C01742=50.626,-85.269,61.037,-178.4250,1.8965,-10229.3015
C01743=46.265,-88.593,61.359,-179.8629,0.0736,-10232.4256
C01744=41.009,-91.197,61.571,-179.9828,0.0078,-10235.7877
C01745=35.488,-93.484,61.571,-179.9823,0.0066,-10239.2124
C01746=29.931,-95.359,61.359,-179.8510,0.0449,-10242.5741
C01747=24.496,-96.092,61.037,-177.5461,-0.2275,-10245.6986
C01748=19.672,-94.474,60.719,-175.8447,-2.5954,-10248.2376
C01749=16.396,-90.884,60.330,-176.4208,-7.1953,-10249.7735
C01750=15.041,-85.905,59.597,-178.1039,-7.6987,-10250.0688
C01751=13.963,-80.549,58.128,-178.6435,-5.7936,-10250.1656
C01752=12.951,-75.822,56.240,-179.3107,-2.5537,-10250.3070
C01753=11.825,-72.328,54.436,178.2362,4.4065,-10250.7148
C01754=9.959,-70.362,53.146,152.3999,15.9321,-10251.9439
C01755=6.412,-69.984,52.637,141.4077,0.6880,-10254.7651
C01756=3.072,-70.158,52.615,141.0087,-2.3123,-10257.4928
C01757=0.000,-70.224,52.630,140.9842,-0.0003,-10260.0000
C01758=0.000,-70.224,52.630,140.9842,-0.0003,-10260.0000
C01759=-3.071,-70.158,52.615,141.0086,2.3125,-10262.5064
C01760=-6.412,-69.984,52.637,141.4081,-0.6906,-10265.2349
C01761=-9.959,-70.362,53.146,152.3995,-15.9318,-10268.0561
C01762=-11.825,-72.328,54.436,178.2362,-4.4065,-10269.2852
C01763=-12.951,-75.822,56.240,-179.3107,2.5537,-10269.6930
C01764=-13.963,-80.549,58.128,-178.6435,5.7936,-10269.8344
C01765=-15.041,-85.905,59.597,-178.1039,7.6987,-10269.9312
C01766=-16.396,-90.884,60.330,-176.4208,7.1953,-10270.2265
C01767=-19.672,-94.474,60.719,-175.8447,2.5954,-10271.7624
C01768=-24.496,-96.092,61.037,-177.5461,0.2275,-10274.3014
C01769=-29.931,-95.359,61.359,-179.8510,-0.0449,-10277.4259
C01770=-35.488,-93.484,61.571,-179.9823,-0.0066,-10280.7876
C01771=-41.009,-91.197,61.571,-179.9828,-0.0078,-10284.2123
C01772=-46.265,-88.593,61.359,-179.8629,-0.0736,-10287.5744
C01773=-50.626,-85.269,61.037,-178.4250,-1.8965,-10290.6985
C01774=-52.893,-80.714,60.719,-178.8932,-4.7688,-10293.2374
C01775=-52.671,-75.858,60.330,177.4212,-7.6040,-10294.7737
C01776=-50.109,-71.379,59.597,175.8716,-6.7862,-10295.0694
C01777=-47.084,-66.830,58.128,176.8518,-5.0569,-10295.1660
C01778=-44.457,-62.772,56.240,178.6807,-2.2931,-10295.3073
C01779=-42.782,-59.505,54.436,-178.1262,4.3612,-10295.7148
C01780=-42.712,-56.796,53.146,170.4736,29.7489,-10296.9441
C01781=-44.952,-54.020,52.637,150.9334,29.8046,-10299.7651
C01782=-47.437,-51.781,52.615,148.9950,28.5406,-10302.4931
C01783=-49.656,-49.656,52.630,150.1903,29.8094,-10305.0000
C01784=-51.781,-47.437,52.615,151.4594,31.0052,-10307.5069
C01785=-54.020,-44.952,52.637,150.1944,29.0648,-10310.2349
C01786=-56.796,-42.711,53.146,150.2510,9.5269,-10313.0566
C01787=-59.505,-42.782,54.436,175.6388,-1.8738,-10314.2852
C01788=-62.772,-44.457,56.240,-177.7069,1.3193,-10314.6927
C01789=-66.830,-47.084,58.128,-174.9431,3.1482,-10314.8340
C01790=-71.379,-50.109,59.597,-173.2138,4.1284,-10314.9306
C01791=-75.858,-52.671,60.330,-172.3960,2.5788,-10315.2263
C01792=-80.714,-52.893,60.719,-175.2312,-1.1068,-10316.7626
C01793=-85.269,-50.626,61.037,-178.1035,-1.5750,-10319.3015
C01794=-88.593,-46.265,61.359,-179.9264,-0.1371,-10322.4256
C01795=-91.197,-41.009,61.571,-179.9922,-0.0172,-10325.7877
C01796=-93.484,-35.488,61.571,-179.9934,-0.0177,-10329.2124
C01797=-95.359,-29.931,61.359,-179.9551,-0.1490,-10332.5741
C01798=-96.092,-24.496,61.037,179.7725,-2.4539,-10335.6986
C01799=-94.474,-19.672,60.719,177.4046,-4.1553,-10338.2376
C01800=-90.884,-16.396,60.330,172.8047,-3.5792,-10339.7735
C01801=-85.905,-15.041,59.597,172.3013,-1.8961,-10340.0688
C01802=-80.549,-13.963,58.128,174.2064,-1.3565,-10340.1656
C01803=-75.822,-12.951,56.240,177.4463,-0.6893,-10340.3070
C01804=-72.328,-11.825,54.436,-175.5935,1.7638,-10340.7148
C01805=-70.362,-9.959,53.146,-164.0679,27.6001,-10341.9439
C01806=-69.984,-6.412,52.637,-179.3120,38.5923,-10344.7651
C01807=-70.158,-3.072,52.615,177.6877,38.9913,-10347.4928
C01808=-70.224,0.000,52.630,179.9997,39.0158,-10350.0000
C01809=-70.158,3.071,52.615,-177.6875,38.9914,-10352.5064
C01810=-69.984,6.412,52.637,179.3094,38.5919,-10355.2349
C01811=-70.362,9.959,53.146,164.0682,27.6005,-10358.0561
C01812=-72.328,11.825,54.436,175.5935,1.7638,-10359.2852
C01813=-75.822,12.951,56.240,-177.4463,-0.6893,-10359.6930
C01814=-80.549,13.963,58.128,-174.2064,-1.3565,-10359.8344
C01815=-85.905,15.041,59.597,-172.3013,-1.8961,-10359.9312
C01816=-90.884,16.396,60.330,-172.8047,-3.5792,-10360.2265
C01817=-94.474,19.672,60.719,-177.4046,-4.1553,-10361.7624
C01818=-96.092,24.496,61.037,-179.7725,-2.4539,-10364.3014
C01819=-95.359,29.931,61.359,179.9551,-0.1490,-10367.4259
C01820=-93.484,35.488,61.571,179.9934,-0.0177,-10370.7876
C01821=-91.197,41.009,61.571,179.9922,-0.0172,-10374.2123
C01822=-88.593,46.265,61.359,179.9264,-0.1371,-10377.5744
C01823=-85.269,50.626,61.037,178.1035,-1.5750,-10380.6985
C01824=-80.714,52.893,60.719,175.2312,-1.1068,-10383.2374
C01825=-75.858,52.671,60.330,172.3960,2.5788,-10384.7737
C01826=-71.379,50.109,59.597,173.2138,4.1284,-10385.0694
C01827=-66.830,47.084,58.128,174.9431,3.1482,-10385.1660
C01828=-62.772,44.457,56.240,177.7069,1.3193,-10385.3073
C01829=-59.505,42.782,54.436,-175.6388,-1.8738,-10385.7148
C01830=-56.796,42.712,53.146,-150.2511,9.5264,-10386.9441
C01831=-54.020,44.952,52.637,-150.1954,29.0666,-10389.7651
C01832=-51.781,47.437,52.615,-151.4594,31.0050,-10392.4931
C01833=-49.656,49.656,52.630,-150.1906,29.8097,-10395.0000
C01834=-47.437,51.781,52.615,-148.9948,28.5406,-10397.5069
C01835=-44.952,54.020,52.637,-150.9352,29.8056,-10400.2349
C01836=-42.711,56.796,53.146,-170.4731,29.7490,-10403.0566
C01837=-42.782,59.505,54.436,178.1262,4.3612,-10404.2852
C01838=-44.457,62.772,56.240,-178.6807,-2.2931,-10404.6927
C01839=-47.084,66.830,58.128,-176.8518,-5.0569,-10404.8340
C01840=-50.109,71.379,59.597,-175.8716,-6.7862,-10404.9306
C01841=-52.671,75.858,60.330,-177.4212,-7.6040,-10405.2263
C01842=-52.893,80.714,60.719,178.8932,-4.7688,-10406.7626
C01843=-50.626,85.269,61.037,178.4250,-1.8965,-10409.3015
C01844=-46.265,88.593,61.359,179.8629,-0.0736,-10412.4256
C01845=-41.009,91.197,61.571,179.9828,-0.0078,-10415.7877
C01846=-35.488,93.484,61.571,179.9823,-0.0066,-10419.2124
C01847=-29.931,95.359,61.359,179.8510,-0.0449,-10422.5741
C01848=-24.496,96.092,61.037,177.5461,0.2275,-10425.6986
C01849=-19.672,94.474,60.719,175.8447,2.5954,-10428.2376
C01850=-16.396,90.884,60.330,176.4208,7.1953,-10429.7735
C01851=-15.041,85.905,59.597,178.1039,7.6987,-10430.0688
C01852=-13.963,80.549,58.128,178.6435,5.7936,-10430.1656
C01853=-12.951,75.822,56.240,179.3107,2.5537,-10430.3070
C01854=-11.825,72.328,54.436,-178.2362,-4.4065,-10430.7148
C01855=-9.959,70.362,53.146,-152.3995,-15.9318,-10431.9439
C01856=-6.412,69.984,52.637,-141.4081,-0.6906,-10434.7651
C01857=-3.071,70.158,52.615,-141.0086,2.3125,-10437.4936
C01858=0.000,70.224,52.630,-140.9842,-0.0003,-10440.0000
C01859=0.000,68.843,54.342,-141.2235,-0.0004,-10440.0000
C01860=2.945,68.781,54.326,-141.2470,-2.2595,-10442.4517
C01861=6.200,68.619,54.350,-141.6907,1.0492,-10445.1629
C01862=9.699,69.044,54.888,-153.6475,16.2162,-10447.9963
C01863=11.507,71.127,56.252,-178.7377,3.4210,-10449.1897
C01864=12.586,74.809,58.158,179.2393,-3.0039,-10449.5501
C01865=13.569,79.780,60.151,178.6797,-5.9734,-10449.6525
C01866=14.621,85.405,61.698,178.2099,-7.7575,-10449.7146
C01867=15.942,90.636,62.469,176.5679,-7.2955,-10449.9757
C01868=19.246,94.423,62.877,175.8470,-2.7058,-10451.5206
C01869=24.159,96.154,63.210,177.5359,-0.2528,-10454.1038
C01870=29.718,95.429,63.547,179.8486,0.0454,-10457.2974
C01871=35.416,93.512,63.770,179.9821,0.0067,-10460.7433
C01872=41.080,91.166,63.770,179.9826,0.0079,-10464.2566
C01873=46.465,88.493,63.547,179.8609,0.0749,-10467.7026
C01874=50.908,85.074,63.210,178.4357,1.9214,-10470.8962
C01875=53.158,80.376,62.877,178.9730,4.8449,-10473.4793
C01876=52.817,75.362,62.469,-177.2451,7.5721,-10475.0245
C01877=50.052,70.729,61.698,-175.7549,6.7538,-10475.2855
C01878=46.818,66.007,60.151,-176.6982,5.1590,-10475.3476
C01879=43.998,61.798,58.158,-178.4123,2.6620,-10475.4495
C01880=42.158,58.431,56.252,178.4711,-3.3109,-10475.8105
C01881=41.963,55.679,54.888,-171.7704,-29.0710,-10477.0038
C01882=44.137,52.905,54.350,-151.3798,-29.7512,-10479.8372
C01883=46.553,50.718,54.326,-149.2273,-28.3546,-10482.5482
C01884=48.679,48.679,54.342,-150.4011,-29.5986,-10485.0000
C01885=50.718,46.553,54.326,-151.6456,-30.7729,-10487.4518
C01886=52.905,44.137,54.350,-150.2477,-28.6184,-10490.1628
C01887=55.680,41.963,54.888,-150.9289,-8.2300,-10492.9966
C01888=58.431,42.158,56.252,-176.6891,1.5289,-10494.1895
C01889=61.798,43.998,58.158,177.3380,-1.5877,-10494.5505
C01890=66.007,46.818,60.151,174.8410,-3.3018,-10494.6524
C01891=70.729,50.052,61.698,173.2462,-4.2451,-10494.7145
C01892=75.362,52.817,62.469,172.4279,-2.7549,-10494.9755
C01893=80.376,53.158,62.877,175.1551,1.0270,-10496.5207
C01894=85.074,50.908,63.210,178.0786,1.5643,-10499.1038
C01895=88.493,46.465,63.547,179.9251,0.1391,-10502.2974
C01896=91.166,41.080,63.770,179.9921,0.0174,-10505.7434
C01897=93.512,35.416,63.770,179.9933,0.0179,-10509.2567
C01898=95.429,29.718,63.547,179.9546,0.1514,-10512.7026
C01899=96.154,24.159,63.210,-179.7472,2.4641,-10515.8962
C01900=94.423,19.246,62.877,-177.2942,4.1530,-10518.4794
C01901=90.636,15.942,62.469,-172.7045,3.4321,-10520.0243
C01902=85.405,14.621,61.698,-172.2425,1.7901,-10520.2854
C01903=79.780,13.569,60.151,-174.0266,1.3203,-10520.3475
C01904=74.809,12.586,58.158,-176.9961,0.7607,-10520.4499
C01905=71.127,11.507,56.252,176.5790,-1.2623,-10520.8103
C01906=69.044,9.699,54.888,163.7838,-26.3525,-10522.0037
C01907=68.619,6.200,54.350,178.9508,-38.3093,-10524.8371
C01908=68.781,2.945,54.326,-177.7405,-38.7530,-10527.5483
C01909=68.843,0.000,54.342,-179.9996,-38.7765,-10530.0000
C01910=68.781,-2.945,54.326,177.7401,-38.7530,-10532.4517
C01911=68.619,-6.200,54.350,-178.9482,-38.3089,-10535.1629
C01912=69.044,-9.699,54.888,-163.7840,-26.3528,-10537.9963
C01913=71.127,-11.507,56.252,-176.5790,-1.2623,-10539.1897
C01914=74.809,-12.586,58.158,176.9961,0.7607,-10539.5501
C01915=79.780,-13.569,60.151,174.0266,1.3203,-10539.6525
C01916=85.405,-14.621,61.698,172.2425,1.7901,-10539.7146
C01917=90.636,-15.942,62.469,172.7045,3.4321,-10539.9757
C01918=94.423,-19.246,62.877,177.2942,4.1530,-10541.5206
C01919=96.154,-24.159,63.210,179.7472,2.4641,-10544.1038
C01920=95.429,-29.718,63.547,-179.9546,0.1514,-10547.2974
C01921=93.512,-35.416,63.770,-179.9933,0.0179,-10550.7433
C01922=91.166,-41.080,63.770,-179.9921,0.0174,-10554.2566
C01923=88.493,-46.465,63.547,-179.9251,0.1391,-10557.7026
C01924=85.074,-50.908,63.210,-178.0786,1.5643,-10560.8962
C01925=80.376,-53.158,62.877,-175.1551,1.0270,-10563.4793
C01926=75.362,-52.817,62.469,-172.4279,-2.7549,-10565.0245
C01927=70.729,-50.052,61.698,-173.2462,-4.2451,-10565.2855
C01928=66.007,-46.818,60.151,-174.8410,-3.3018,-10565.3476
C01929=61.798,-43.998,58.158,-177.3380,-1.5877,-10565.4495
C01930=58.431,-42.158,56.252,176.6891,1.5289,-10565.8105
C01931=55.679,-41.963,54.888,150.9290,-8.2296,-10567.0038
C01932=52.905,-44.137,54.350,150.2488,-28.6202,-10569.8372
C01933=50.718,-46.553,54.326,151.6454,-30.7727,-10572.5482
C01934=48.679,-48.679,54.342,150.4014,-29.5989,-10575.0000
C01935=46.553,-50.718,54.326,149.2271,-28.3544,-10577.4518
C01936=44.137,-52.905,54.350,151.3816,-29.7523,-10580.1628
C01937=41.963,-55.680,54.888,171.7700,-29.0711,-10582.9966
C01938=42.158,-58.431,56.252,-178.4711,-3.3109,-10584.1895
C01939=43.998,-61.798,58.158,178.4123,2.6620,-10584.5505
C01940=46.818,-66.007,60.151,176.6982,5.1590,-10584.6524
C01941=50.052,-70.729,61.698,175.7549,6.7538,-10584.7145
C01942=52.817,-75.362,62.469,177.2451,7.5721,-10584.9755
C01943=53.158,-80.376,62.877,-178.9730,4.8449,-10586.5207
C01944=50.908,-85.074,63.210,-178.4357,1.9214,-10589.1038
C01945=46.465,-88.493,63.547,-179.8609,0.0749,-10592.2974
C01946=41.080,-91.166,63.770,-179.9826,0.0079,-10595.7434
C01947=35.416,-93.512,63.770,-179.9821,0.0067,-10599.2567
C01948=29.718,-95.429,63.547,-179.8486,0.0454,-10602.7026
C01949=24.159,-96.154,63.210,-177.5359,-0.2528,-10605.8962
C01950=19.246,-94.423,62.877,-175.8470,-2.7058,-10608.4794
C01951=15.942,-90.636,62.469,-176.5679,-7.2955,-10610.0243
C01952=14.621,-85.405,61.698,-178.2099,-7.7575,-10610.2854
C01953=13.569,-79.780,60.151,-178.6797,-5.9734,-10610.3475
C01954=12.586,-74.809,58.158,-179.2393,-3.0039,-10610.4499
C01955=11.507,-71.127,56.252,178.7377,3.4210,-10610.8103
C01956=9.699,-69.044,54.888,153.6475,16.2162,-10612.0037
C01957=6.200,-68.619,54.350,141.6907,1.0492,-10614.8371
C01958=2.945,-68.781,54.326,141.2470,-2.2595,-10617.5483
C01959=0.000,-68.843,54.342,141.2235,-0.0004,-10620.0000
C01960=0.000,-68.843,54.342,141.2235,-0.0004,-10620.0000
C01961=-2.945,-68.781,54.326,141.2470,2.2599,-10622.4517
C01962=-6.200,-68.619,54.350,141.6911,-1.0518,-10625.1629
C01963=-9.699,-69.044,54.888,153.6472,-16.2160,-10627.9963
C01964=-11.507,-71.127,56.252,178.7377,-3.4210,-10629.1897
C01965=-12.586,-74.809,58.158,-179.2393,3.0039,-10629.5501
C01966=-13.569,-79.780,60.151,-178.6797,5.9734,-10629.6525
C01967=-14.621,-85.405,61.698,-178.2099,7.7575,-10629.7146
C01968=-15.942,-90.636,62.469,-176.5679,7.2955,-10629.9757
C01969=-19.246,-94.423,62.877,-175.8470,2.7058,-10631.5206
C01970=-24.159,-96.154,63.210,-177.5359,0.2528,-10634.1038
C01971=-29.718,-95.429,63.547,-179.8486,-0.0454,-10637.2974
C01972=-35.416,-93.512,63.770,-179.9821,-0.0067,-10640.7433
C01973=-41.080,-91.166,63.770,-179.9826,-0.0079,-10644.2566
C01974=-46.465,-88.493,63.547,-179.8609,-0.0749,-10647.7026
C01975=-50.908,-85.074,63.210,-178.4357,-1.9214,-10650.8962
C01976=-53.158,-80.376,62.877,-178.9730,-4.8449,-10653.4793
C01977=-52.817,-75.362,62.469,177.2451,-7.5721,-10655.0245
C01978=-50.052,-70.729,61.698,175.7549,-6.7538,-10655.2855
C01979=-46.818,-66.007,60.151,176.6982,-5.1590,-10655.3476
C01980=-43.998,-61.798,58.158,178.4123,-2.6620,-10655.4495
C01981=-42.158,-58.431,56.252,-178.4711,3.3109,-10655.8105
C01982=-41.963,-55.679,54.888,171.7704,29.0710,-10657.0038
C01983=-44.137,-52.905,54.350,151.3798,29.7512,-10659.8372
C01984=-46.553,-50.718,54.326,149.2273,28.3546,-10662.5482
C01985=-48.679,-48.679,54.342,150.4011,29.5986,-10665.0000
C01986=-50.718,-46.553,54.326,151.6456,30.7729,-10667.4518
C01987=-52.905,-44.137,54.350,150.2477,28.6184,-10670.1628
C01988=-55.680,-41.963,54.888,150.9289,8.2300,-10672.9966
C01989=-58.431,-42.158,56.252,176.6891,-1.5289,-10674.1895
C01990=-61.798,-43.998,58.158,-177.3380,1.5877,-10674.5505
C01991=-66.007,-46.818,60.151,-174.8410,3.3018,-10674.6524
C01992=-70.729,-50.052,61.698,-173.2462,4.2451,-10674.7145
C01993=-75.362,-52.817,62.469,-172.4279,2.7549,-10674.9755
C01994=-80.376,-53.158,62.877,-175.1551,-1.0270,-10676.5207
C01995=-85.074,-50.908,63.210,-178.0786,-1.5643,-10679.1038
C01996=-88.493,-46.465,63.547,-179.9251,-0.1391,-10682.2974
C01997=-91.166,-41.080,63.770,-179.9921,-0.0174,-10685.7434
C01998=-93.512,-35.416,63.770,-179.9933,-0.0179,-10689.2567
C01999=-95.429,-29.718,63.547,-179.9546,-0.1514,-10692.7026
///TOOL 0
///POSTYPE ANGLE
///ANGLE
EC00000=0.0000,7126.2037
EC00001=0.0000,7128.6701
EC00002=0.0000,7131.2180
EC00003=0.0000,7133.7821
EC00004=0.0000,7136.3297
EC00005=0.0000,7138.7961
EC00006=0.0000,7140.9450
EC00007=0.0000,7142.4587
EC00008=0.0000,7143.1487
EC00009=0.0000,7143.6320
EC00010=0.0000,7144.1614
EC00011=0.0000,7144.9722
EC00012=0.0000,7146.4919
EC00013=0.0000,7149.2230
EC00014=0.0000,7152.0820
EC00015=0.0000,7155.0000
EC00016=0.0000,7157.9180
EC00017=0.0000,7160.7770
EC00018=0.0000,7163.5081
EC00019=0.0000,7165.0278
EC00020=0.0000,7165.8386
EC00021=0.0000,7166.3680
EC00022=0.0000,7166.8513
EC00023=0.0000,7167.5413
EC00024=0.0000,7169.0550
EC00025=0.0000,7171.2039
EC00026=0.0000,7173.6703
EC00027=0.0000,7176.2179
EC00028=0.0000,7178.7820
EC00029=0.0000,7181.3299
EC00030=0.0000,7183.7963
EC00031=0.0000,7185.9450
EC00032=0.0000,7187.4590
EC00033=0.0000,7188.1488
EC00034=0.0000,7188.6317
EC00035=0.0000,7189.1618
EC00036=0.0000,7189.9720
EC00037=0.0000,7191.4924
EC00038=0.0000,7194.2225
EC00039=0.0000,7197.0820
EC00040=0.0000,7200.0000
EC00041=0.0000,7200.0000
EC00042=0.0000,7202.8792
EC00043=0.0000,7205.7259
EC00044=0.0000,7208.4654
EC00045=0.0000,7209.9566
EC00046=0.0000,7210.7254
EC00047=0.0000,7211.2119
EC00048=0.0000,7211.6495
EC00049=0.0000,7212.2909
EC00050=0.0000,7213.8024
EC00051=0.0000,7215.9922
EC00052=0.0000,7218.5312
EC00053=0.0000,7221.1696
EC00054=0.0000,7223.8303
EC00055=0.0000,7226.4689
EC00056=0.0000,7229.0082
EC00057=0.0000,7231.1977
EC00058=0.0000,7232.7089
EC00059=0.0000,7233.3509
EC00060=0.0000,7233.7878
EC00061=0.0000,7234.2746
EC00062=0.0000,7235.0436
EC00063=0.0000,7236.5348
EC00064=0.0000,7239.2737
EC00065=0.0000,7242.1206
EC00066=0.0000,7245.0000
EC00067=0.0000,7247.8789
EC00068=0.0000,7250.7263
EC00069=0.0000,7253.4652
EC00070=0.0000,7254.9564
EC00071=0.0000,7255.7254
EC00072=0.0000,7256.2122
EC00073=0.0000,7256.6491
EC00074=0.0000,7257.2911
EC00075=0.0000,7258.8023
EC00076=0.0000,7260.9918
EC00077=0.0000,7263.5311
EC00078=0.0000,7266.1697
EC00079=0.0000,7268.8304
EC00080=0.0000,7271.4688
EC00081=0.0000,7274.0078
EC00082=0.0000,7276.1976
EC00083=0.0000,7277.7091
EC00084=0.0000,7278.3505
EC00085=0.0000,7278.7881
EC00086=0.0000,7279.2746
EC00087=0.0000,7280.0434
EC00088=0.0000,7281.5346
EC00089=0.0000,7284.2741
EC00090=0.0000,7287.1208
EC00091=0.0000,7290.0000
EC00092=0.0000,7292.8792
EC00093=0.0000,7295.7266
EC00094=0.0000,7298.4654
EC00095=0.0000,7299.9566
EC00096=0.0000,7300.7254
EC00097=0.0000,7301.2119
EC00098=0.0000,7301.6495
EC00099=0.0000,7302.2909
EC00100=0.0000,7303.8024
EC00101=0.0000,7305.9922
EC00102=0.0000,7308.5312
EC00103=0.0000,7311.1696
EC00104=0.0000,7313.8303
EC00105=0.0000,7316.4689
EC00106=0.0000,7319.0082
EC00107=0.0000,7321.1977
EC00108=0.0000,7322.7089
EC00109=0.0000,7323.3509
EC00110=0.0000,7323.7878
EC00111=0.0000,7324.2746
EC00112=0.0000,7325.0436
EC00113=0.0000,7326.5348
EC00114=0.0000,7329.2737
EC00115=0.0000,7332.1206
EC00116=0.0000,7335.0000
EC00117=0.0000,7337.8789
EC00118=0.0000,7340.7263
EC00119=0.0000,7343.4652
EC00120=0.0000,7344.9564
EC00121=0.0000,7345.7254
EC00122=0.0000,7346.2122
EC00123=0.0000,7346.6491
EC00124=0.0000,7347.2911
EC00125=0.0000,7348.8023
EC00126=0.0000,7350.9918
EC00127=0.0000,7353.5311
EC00128=0.0000,7356.1697
EC00129=0.0000,7358.8304
EC00130=0.0000,7361.4688
EC00131=0.0000,7364.0078
EC00132=0.0000,7366.1976
EC00133=0.0000,7367.7091
EC00134=0.0000,7368.3505
EC00135=0.0000,7368.7881
EC00136=0.0000,7369.2746
EC00137=0.0000,7370.0434
EC00138=0.0000,7371.5346
EC00139=0.0000,7374.2741
EC00140=0.0000,7377.1208
EC00141=0.0000,7380.0000
EC00142=0.0000,7380.0000
EC00143=0.0000,7382.8792
EC00144=0.0000,7385.7266
EC00145=0.0000,7388.4654
EC00146=0.0000,7389.9566
EC00147=0.0000,7390.7254
EC00148=0.0000,7391.2119
EC00149=0.0000,7391.6495
EC00150=0.0000,7392.2909
EC00151=0.0000,7393.8024
EC00152=0.0000,7395.9922
EC00153=0.0000,7398.5312
EC00154=0.0000,7401.1696
EC00155=0.0000,7403.8303
EC00156=0.0000,7406.4689
EC00157=0.0000,7409.0082
EC00158=0.0000,7411.1977
EC00159=0.0000,7412.7089
EC00160=0.0000,7413.3509
EC00161=0.0000,7413.7878
EC00162=0.0000,7414.2746
EC00163=0.0000,7415.0436
EC00164=0.0000,7416.5348
EC00165=0.0000,7419.2737
EC00166=0.0000,7422.1206
EC00167=0.0000,7425.0000
EC00168=0.0000,7427.8789
EC00169=0.0000,7430.7263
EC00170=0.0000,7433.4652
EC00171=0.0000,7434.9564
EC00172=0.0000,7435.7254
EC00173=0.0000,7436.2122
EC00174=0.0000,7436.6491
EC00175=0.0000,7437.2911
EC00176=0.0000,7438.8023
EC00177=0.0000,7440.9918
EC00178=0.0000,7443.5311
EC00179=0.0000,7446.1697
EC00180=0.0000,7448.8304
EC00181=0.0000,7451.4688
EC00182=0.0000,7454.0078
EC00183=0.0000,7456.1976
EC00184=0.0000,7457.7091
EC00185=0.0000,7458.3505
EC00186=0.0000,7458.7881
EC00187=0.0000,7459.2746
EC00188=0.0000,7460.0434
EC00189=0.0000,7461.5346
EC00190=0.0000,7464.2741
EC00191=0.0000,7467.1208
EC00192=0.0000,7470.0000
EC00193=0.0000,7472.8792
EC00194=0.0000,7475.7266
EC00195=0.0000,7478.4654
EC00196=0.0000,7479.9566
EC00197=0.0000,7480.7254
EC00198=0.0000,7481.2119
EC00199=0.0000,7481.6495
EC00200=0.0000,7482.2909
EC00201=0.0000,7483.8024
EC00202=0.0000,7485.9922
EC00203=0.0000,7488.5312
EC00204=0.0000,7491.1696
EC00205=0.0000,7493.8303
EC00206=0.0000,7496.4689
EC00207=0.0000,7499.0082
EC00208=0.0000,7501.1977
EC00209=0.0000,7502.7089
EC00210=0.0000,7503.3509
EC00211=0.0000,7503.7878
EC00212=0.0000,7504.2746
EC00213=0.0000,7505.0436
EC00214=0.0000,7506.5348
EC00215=0.0000,7509.2737
EC00216=0.0000,7512.1206
EC00217=0.0000,7515.0000
EC00218=0.0000,7517.8789
EC00219=0.0000,7520.7263
EC00220=0.0000,7523.4652
EC00221=0.0000,7524.9564
EC00222=0.0000,7525.7254
EC00223=0.0000,7526.2122
EC00224=0.0000,7526.6491
EC00225=0.0000,7527.2911
EC00226=0.0000,7528.8023
EC00227=0.0000,7530.9918
EC00228=0.0000,7533.5311
EC00229=0.0000,7536.1697
EC00230=0.0000,7538.8304
EC00231=0.0000,7541.4688
EC00232=0.0000,7544.0078
EC00233=0.0000,7546.1976
EC00234=0.0000,7547.7091
EC00235=0.0000,7548.3505
EC00236=0.0000,7548.7881
EC00237=0.0000,7549.2746
EC00238=0.0000,7550.0434
EC00239=0.0000,7551.5346
EC00240=0.0000,7554.2734
EC00241=0.0000,7557.1208
EC00242=0.0000,7560.0000
EC00243=0.0000,7560.0000
EC00244=0.0000,7562.8388
EC00245=0.0000,7565.6728
EC00246=0.0000,7568.4202
EC00247=0.0000,7569.8823
EC00248=0.0000,7570.6084
EC00249=0.0000,7571.0516
EC00250=0.0000,7571.4429
EC00251=0.0000,7572.0370
EC00252=0.0000,7573.5473
EC00253=0.0000,7575.7781
EC00254=0.0000,7578.3907
EC00255=0.0000,7581.1209
EC00256=0.0000,7583.8793
EC00257=0.0000,7586.6097
EC00258=0.0000,7589.2218
EC00259=0.0000,7591.4529
EC00260=0.0000,7592.9628
EC00261=0.0000,7593.5569
EC00262=0.0000,7593.9481
EC00263=0.0000,7594.3909
EC00264=0.0000,7595.1173
EC00265=0.0000,7596.5793
EC00266=0.0000,7599.3269
EC00267=0.0000,7602.1606
EC00268=0.0000,7605.0000
EC00269=0.0000,7607.8388
EC00270=0.0000,7610.6731
EC00271=0.0000,7613.4207
EC00272=0.0000,7614.8827
EC00273=0.0000,7615.6091
EC00274=0.0000,7616.0519
EC00275=0.0000,7616.4431
EC00276=0.0000,7617.0372
EC00277=0.0000,7618.5471
EC00278=0.0000,7620.7782
EC00279=0.0000,7623.3903
EC00280=0.0000,7626.1207
EC00281=0.0000,7628.8791
EC00282=0.0000,7631.6093
EC00283=0.0000,7634.2219
EC00284=0.0000,7636.4527
EC00285=0.0000,7637.9630
EC00286=0.0000,7638.5571
EC00287=0.0000,7638.9484
EC00288=0.0000,7639.3916
EC00289=0.0000,7640.1177
EC00290=0.0000,7641.5798
EC00291=0.0000,7644.3272
EC00292=0.0000,7647.1612
EC00293=0.0000,7650.0000
EC00294=0.0000,7652.8388
EC00295=0.0000,7655.6728
EC00296=0.0000,7658.4209
EC00297=0.0000,7659.8823
EC00298=0.0000,7660.6084
EC00299=0.0000,7661.0516
EC00300=0.0000,7661.4429
EC00301=0.0000,7662.0370
EC00302=0.0000,7663.5473
EC00303=0.0000,7665.7781
EC00304=0.0000,7668.3907
EC00305=0.0000,7671.1209
EC00306=0.0000,7673.8793
EC00307=0.0000,7676.6097
EC00308=0.0000,7679.2218
EC00309=0.0000,7681.4529
EC00310=0.0000,7682.9628
EC00311=0.0000,7683.5569
EC00312=0.0000,7683.9481
EC00313=0.0000,7684.3909
EC00314=0.0000,7685.1173
EC00315=0.0000,7686.5793
EC00316=0.0000,7689.3269
EC00317=0.0000,7692.1606
EC00318=0.0000,7695.0000
EC00319=0.0000,7697.8388
EC00320=0.0000,7700.6731
EC00321=0.0000,7703.4207
EC00322=0.0000,7704.8827
EC00323=0.0000,7705.6091
EC00324=0.0000,7706.0519
EC00325=0.0000,7706.4431
EC00326=0.0000,7707.0372
EC00327=0.0000,7708.5471
EC00328=0.0000,7710.7782
EC00329=0.0000,7713.3903
EC00330=0.0000,7716.1207
EC00331=0.0000,7718.8791
EC00332=0.0000,7721.6093
EC00333=0.0000,7724.2219
EC00334=0.0000,7726.4527
EC00335=0.0000,7727.9630
EC00336=0.0000,7728.5571
EC00337=0.0000,7728.9484
EC00338=0.0000,7729.3916
EC00339=0.0000,7730.1177
EC00340=0.0000,7731.5798
EC00341=0.0000,7734.3272
EC00342=0.0000,7737.1612
EC00343=0.0000,7740.0000
EC00344=0.0000,7740.0000
EC00345=0.0000,7742.8388
EC00346=0.0000,7745.6728
EC00347=0.0000,7748.4209
EC00348=0.0000,7749.8823
EC00349=0.0000,7750.6084
EC00350=0.0000,7751.0516
EC00351=0.0000,7751.4429
EC00352=0.0000,7752.0370
EC00353=0.0000,7753.5473
EC00354=0.0000,7755.7781
EC00355=0.0000,7758.3907
EC00356=0.0000,7761.1209
EC00357=0.0000,7763.8793
EC00358=0.0000,7766.6097
EC00359=0.0000,7769.2218
EC00360=0.0000,7771.4529
EC00361=0.0000,7772.9628
EC00362=0.0000,7773.5569
EC00363=0.0000,7773.9481
EC00364=0.0000,7774.3909
EC00365=0.0000,7775.1173
EC00366=0.0000,7776.5793
EC00367=0.0000,7779.3269
EC00368=0.0000,7782.1606
EC00369=0.0000,7785.0000
EC00370=0.0000,7787.8388
EC00371=0.0000,7790.6731
EC00372=0.0000,7793.4207
EC00373=0.0000,7794.8827
EC00374=0.0000,7795.6091
EC00375=0.0000,7796.0519
EC00376=0.0000,7796.4431
EC00377=0.0000,7797.0372
EC00378=0.0000,7798.5471
EC00379=0.0000,7800.7782
EC00380=0.0000,7803.3903
EC00381=0.0000,7806.1207
EC00382=0.0000,7808.8791
EC00383=0.0000,7811.6093
EC00384=0.0000,7814.2219
EC00385=0.0000,7816.4527
EC00386=0.0000,7817.9630
EC00387=0.0000,7818.5571
EC00388=0.0000,7818.9484
EC00389=0.0000,7819.3916
EC00390=0.0000,7820.1177
EC00391=0.0000,7821.5798
EC00392=0.0000,7824.3272
EC00393=0.0000,7827.1612
EC00394=0.0000,7830.0000
EC00395=0.0000,7832.8388
EC00396=0.0000,7835.6728
EC00397=0.0000,7838.4209
EC00398=0.0000,7839.8823
EC00399=0.0000,7840.6084
EC00400=0.0000,7841.0516
EC00401=0.0000,7841.4429
EC00402=0.0000,7842.0370
EC00403=0.0000,7843.5473
EC00404=0.0000,7845.7781
EC00405=0.0000,7848.3907
EC00406=0.0000,7851.1209
EC00407=0.0000,7853.8793
EC00408=0.0000,7856.6097
EC00409=0.0000,7859.2218
EC00410=0.0000,7861.4529
EC00411=0.0000,7862.9628
EC00412=0.0000,7863.5569
EC00413=0.0000,7863.9481
EC00414=0.0000,7864.3909
EC00415=0.0000,7865.1173
EC00416=0.0000,7866.5793
EC00417=0.0000,7869.3269
EC00418=0.0000,7872.1606
EC00419=0.0000,7875.0000
EC00420=0.0000,7877.8388
EC00421=0.0000,7880.6731
EC00422=0.0000,7883.4207
EC00423=0.0000,7884.8827
EC00424=0.0000,7885.6091
EC00425=0.0000,7886.0519
EC00426=0.0000,7886.4431
EC00427=0.0000,7887.0372
EC00428=0.0000,7888.5471
EC00429=0.0000,7890.7782
EC00430=0.0000,7893.3903
EC00431=0.0000,7896.1207
EC00432=0.0000,7898.8791
EC00433=0.0000,7901.6093
EC00434=0.0000,7904.2219
EC00435=0.0000,7906.4527
EC00436=0.0000,7907.9630
EC00437=0.0000,7908.5571
EC00438=0.0000,7908.9484
EC00439=0.0000,7909.3916
EC00440=0.0000,7910.1177
EC00441=0.0000,7911.5791
EC00442=0.0000,7914.3272
EC00443=0.0000,7917.1612
EC00444=0.0000,7920.0000
EC00445=0.0000,7920.0000
EC00446=0.0000,7922.7966
EC00447=0.0000,7925.6177
EC00448=0.0000,7928.3745
EC00449=0.0000,7929.8055
EC00450=0.0000,7930.4884
EC00451=0.0000,7930.8872
EC00452=0.0000,7931.2331
EC00453=0.0000,7931.7800
EC00454=0.0000,7933.2896
EC00455=0.0000,7935.5634
EC00456=0.0000,7938.2498
EC00457=0.0000,7941.0723
EC00458=0.0000,7943.9275
EC00459=0.0000,7946.7502
EC00460=0.0000,7949.4368
EC00461=0.0000,7951.7100
EC00462=0.0000,7953.2198
EC00463=0.0000,7953.7669
EC00464=0.0000,7954.1127
EC00465=0.0000,7954.5119
EC00466=0.0000,7955.1948
EC00467=0.0000,7956.6259
EC00468=0.0000,7959.3828
EC00469=0.0000,7962.2032
EC00470=0.0000,7965.0000
EC00471=0.0000,7967.7968
EC00472=0.0000,7970.6172
EC00473=0.0000,7973.3741
EC00474=0.0000,7974.8052
EC00475=0.0000,7975.4881
EC00476=0.0000,7975.8873
EC00477=0.0000,7976.2331
EC00478=0.0000,7976.7802
EC00479=0.0000,7978.2900
EC00480=0.0000,7980.5632
EC00481=0.0000,7983.2498
EC00482=0.0000,7986.0725
EC00483=0.0000,7988.9277
EC00484=0.0000,7991.7502
EC00485=0.0000,7994.4366
EC00486=0.0000,7996.7104
EC00487=0.0000,7998.2200
EC00488=0.0000,7998.7669
EC00489=0.0000,7999.1128
EC00490=0.0000,7999.5116
EC00491=0.0000,8000.1945
EC00492=0.0000,8001.6255
EC00493=0.0000,8004.3823
EC00494=0.0000,8007.2034
EC00495=0.0000,8010.0000
EC00496=0.0000,8012.7966
EC00497=0.0000,8015.6177
EC00498=0.0000,8018.3745
EC00499=0.0000,8019.8055
EC00500=0.0000,8020.4884
EC00501=0.0000,8020.8872
EC00502=0.0000,8021.2331
EC00503=0.0000,8021.7800
EC00504=0.0000,8023.2896
EC00505=0.0000,8025.5634
EC00506=0.0000,8028.2498
EC00507=0.0000,8031.0723
EC00508=0.0000,8033.9275
EC00509=0.0000,8036.7502
EC00510=0.0000,8039.4368
EC00511=0.0000,8041.7100
EC00512=0.0000,8043.2198
EC00513=0.0000,8043.7669
EC00514=0.0000,8044.1127
EC00515=0.0000,8044.5119
EC00516=0.0000,8045.1948
EC00517=0.0000,8046.6259
EC00518=0.0000,8049.3828
EC00519=0.0000,8052.2032
EC00520=0.0000,8055.0000
EC00521=0.0000,8057.7968
EC00522=0.0000,8060.6172
EC00523=0.0000,8063.3741
EC00524=0.0000,8064.8052
EC00525=0.0000,8065.4881
EC00526=0.0000,8065.8873
EC00527=0.0000,8066.2331
EC00528=0.0000,8066.7802
EC00529=0.0000,8068.2900
EC00530=0.0000,8070.5632
EC00531=0.0000,8073.2498
EC00532=0.0000,8076.0725
EC00533=0.0000,8078.9277
EC00534=0.0000,8081.7502
EC00535=0.0000,8084.4366
EC00536=0.0000,8086.7104
EC00537=0.0000,8088.2200
EC00538=0.0000,8088.7669
EC00539=0.0000,8089.1128
EC00540=0.0000,8089.5116
EC00541=0.0000,8090.1945
EC00542=0.0000,8091.6255
EC00543=0.0000,8094.3823
EC00544=0.0000,8097.2034
EC00545=0.0000,8100.0000
EC00546=0.0000,8100.0000
EC00547=0.0000,8102.7966
EC00548=0.0000,8105.6177
EC00549=0.0000,8108.3745
EC00550=0.0000,8109.8055
EC00551=0.0000,8110.4884
EC00552=0.0000,8110.8872
EC00553=0.0000,8111.2331
EC00554=0.0000,8111.7800
EC00555=0.0000,8113.2896
EC00556=0.0000,8115.5634
EC00557=0.0000,8118.2498
EC00558=0.0000,8121.0723
EC00559=0.0000,8123.9275
EC00560=0.0000,8126.7502
EC00561=0.0000,8129.4368
EC00562=0.0000,8131.7100
EC00563=0.0000,8133.2198
EC00564=0.0000,8133.7669
EC00565=0.0000,8134.1127
EC00566=0.0000,8134.5119
EC00567=0.0000,8135.1948
EC00568=0.0000,8136.6259
EC00569=0.0000,8139.3828
EC00570=0.0000,8142.2032
EC00571=0.0000,8145.0000
EC00572=0.0000,8147.7968
EC00573=0.0000,8150.6172
EC00574=0.0000,8153.3741
EC00575=0.0000,8154.8052
EC00576=0.0000,8155.4881
EC00577=0.0000,8155.8873
EC00578=0.0000,8156.2331
EC00579=0.0000,8156.7802
EC00580=0.0000,8158.2900
EC00581=0.0000,8160.5632
EC00582=0.0000,8163.2498
EC00583=0.0000,8166.0725
EC00584=0.0000,8168.9277
EC00585=0.0000,8171.7502
EC00586=0.0000,8174.4366
EC00587=0.0000,8176.7104
EC00588=0.0000,8178.2200
EC00589=0.0000,8178.7669
EC00590=0.0000,8179.1128
EC00591=0.0000,8179.5116
EC00592=0.0000,8180.1945
EC00593=0.0000,8181.6255
EC00594=0.0000,8184.3823
EC00595=0.0000,8187.2034
EC00596=0.0000,8190.0000
EC00597=0.0000,8192.7966
EC00598=0.0000,8195.6177
EC00599=0.0000,8198.3745
EC00600=0.0000,8199.8055
EC00601=0.0000,8200.4884
EC00602=0.0000,8200.8872
EC00603=0.0000,8201.2331
EC00604=0.0000,8201.7800
EC00605=0.0000,8203.2896
EC00606=0.0000,8205.5634
EC00607=0.0000,8208.2498
EC00608=0.0000,8211.0723
EC00609=0.0000,8213.9275
EC00610=0.0000,8216.7502
EC00611=0.0000,8219.4368
EC00612=0.0000,8221.7100
EC00613=0.0000,8223.2198
EC00614=0.0000,8223.7669
EC00615=0.0000,8224.1127
EC00616=0.0000,8224.5119
EC00617=0.0000,8225.1948
EC00618=0.0000,8226.6259
EC00619=0.0000,8229.3828
EC00620=0.0000,8232.2032
EC00621=0.0000,8235.0000
EC00622=0.0000,8237.7968
EC00623=0.0000,8240.6172
EC00624=0.0000,8243.3741
EC00625=0.0000,8244.8052
EC00626=0.0000,8245.4881
EC00627=0.0000,8245.8873
EC00628=0.0000,8246.2331
EC00629=0.0000,8246.7802
EC00630=0.0000,8248.2900
EC00631=0.0000,8250.5632
EC00632=0.0000,8253.2498
EC00633=0.0000,8256.0725
EC00634=0.0000,8258.9277
EC00635=0.0000,8261.7502
EC00636=0.0000,8264.4366
EC00637=0.0000,8266.7104
EC00638=0.0000,8268.2200
EC00639=0.0000,8268.7669
EC00640=0.0000,8269.1128
EC00641=0.0000,8269.5116
EC00642=0.0000,8270.1945
EC00643=0.0000,8271.6255
EC00644=0.0000,8274.3823
EC00645=0.0000,8277.2034
EC00646=0.0000,8280.0000
EC00647=0.0000,8280.0000
EC00648=0.0000,8282.7531
EC00649=0.0000,8285.5598
EC00650=0.0000,8288.3257
EC00651=0.0000,8289.7254
EC00652=0.0000,8290.3637
EC00653=0.0000,8290.7187
EC00654=0.0000,8291.0200
EC00655=0.0000,8291.5211
EC00656=0.0000,8293.0317
EC00657=0.0000,8295.3479
EC00658=0.0000,8298.1086
EC00659=0.0000,8301.0234
EC00660=0.0000,8303.9765
EC00661=0.0000,8306.8914
EC00662=0.0000,8309.6519
EC00663=0.0000,8311.9680
EC00664=0.0000,8313.4791
EC00665=0.0000,8313.9803
EC00666=0.0000,8314.2813
EC00667=0.0000,8314.6359
EC00668=0.0000,8315.2745
EC00669=0.0000,8316.6744
EC00670=0.0000,8319.4401
EC00671=0.0000,8322.2471
EC00672=0.0000,8325.0000
EC00673=0.0000,8327.7529
EC00674=0.0000,8330.5599
EC00675=0.0000,8333.3256
EC00676=0.0000,8334.7255
EC00677=0.0000,8335.3641
EC00678=0.0000,8335.7187
EC00679=0.0000,8336.0197
EC00680=0.0000,8336.5209
EC00681=0.0000,8338.0320
EC00682=0.0000,8340.3481
EC00683=0.0000,8343.1086
EC00684=0.0000,8346.0235
EC00685=0.0000,8348.9766
EC00686=0.0000,8351.8914
EC00687=0.0000,8354.6521
EC00688=0.0000,8356.9683
EC00689=0.0000,8358.4789
EC00690=0.0000,8358.9800
EC00691=0.0000,8359.2813
EC00692=0.0000,8359.6363
EC00693=0.0000,8360.2746
EC00694=0.0000,8361.6743
EC00695=0.0000,8364.4402
EC00696=0.0000,8367.2469
EC00697=0.0000,8370.0000
EC00698=0.0000,8372.7531
EC00699=0.0000,8375.5598
EC00700=0.0000,8378.3257
EC00701=0.0000,8379.7254
EC00702=0.0000,8380.3637
EC00703=0.0000,8380.7187
EC00704=0.0000,8381.0200
EC00705=0.0000,8381.5211
EC00706=0.0000,8383.0317
EC00707=0.0000,8385.3479
EC00708=0.0000,8388.1086
EC00709=0.0000,8391.0234
EC00710=0.0000,8393.9765
EC00711=0.0000,8396.8914
EC00712=0.0000,8399.6519
EC00713=0.0000,8401.9680
EC00714=0.0000,8403.4791
EC00715=0.0000,8403.9803
EC00716=0.0000,8404.2813
EC00717=0.0000,8404.6359
EC00718=0.0000,8405.2745
EC00719=0.0000,8406.6744
EC00720=0.0000,8409.4401
EC00721=0.0000,8412.2471
EC00722=0.0000,8415.0000
EC00723=0.0000,8417.7529
EC00724=0.0000,8420.5599
EC00725=0.0000,8423.3256
EC00726=0.0000,8424.7255
EC00727=0.0000,8425.3641
EC00728=0.0000,8425.7187
EC00729=0.0000,8426.0197
EC00730=0.0000,8426.5209
EC00731=0.0000,8428.0320
EC00732=0.0000,8430.3481
EC00733=0.0000,8433.1086
EC00734=0.0000,8436.0235
EC00735=0.0000,8438.9766
EC00736=0.0000,8441.8914
EC00737=0.0000,8444.6521
EC00738=0.0000,8446.9683
EC00739=0.0000,8448.4789
EC00740=0.0000,8448.9800
EC00741=0.0000,8449.2813
EC00742=0.0000,8449.6363
EC00743=0.0000,8450.2746
EC00744=0.0000,8451.6743
EC00745=0.0000,8454.4402
EC00746=0.0000,8457.2469
EC00747=0.0000,8460.0000
EC00748=0.0000,8460.0000
EC00749=0.0000,8462.7531
EC00750=0.0000,8465.5598
EC00751=0.0000,8468.3257
EC00752=0.0000,8469.7254
EC00753=0.0000,8470.3637
EC00754=0.0000,8470.7187
EC00755=0.0000,8471.0200
EC00756=0.0000,8471.5211
EC00757=0.0000,8473.0317
EC00758=0.0000,8475.3479
EC00759=0.0000,8478.1086
EC00760=0.0000,8481.0234
EC00761=0.0000,8483.9765
EC00762=0.0000,8486.8914
EC00763=0.0000,8489.6519
EC00764=0.0000,8491.9680
EC00765=0.0000,8493.4791
EC00766=0.0000,8493.9803
EC00767=0.0000,8494.2813
EC00768=0.0000,8494.6359
EC00769=0.0000,8495.2745
EC00770=0.0000,8496.6744
EC00771=0.0000,8499.4401
EC00772=0.0000,8502.2471
EC00773=0.0000,8505.0000
EC00774=0.0000,8507.7529
EC00775=0.0000,8510.5599
EC00776=0.0000,8513.3256
EC00777=0.0000,8514.7255
EC00778=0.0000,8515.3641
EC00779=0.0000,8515.7187
EC00780=0.0000,8516.0197
EC00781=0.0000,8516.5209
EC00782=0.0000,8518.0320
EC00783=0.0000,8520.3481
EC00784=0.0000,8523.1086
EC00785=0.0000,8526.0235
EC00786=0.0000,8528.9766
EC00787=0.0000,8531.8914
EC00788=0.0000,8534.6521
EC00789=0.0000,8536.9683
EC00790=0.0000,8538.4789
EC00791=0.0000,8538.9800
EC00792=0.0000,8539.2813
EC00793=0.0000,8539.6363
EC00794=0.0000,8540.2746
EC00795=0.0000,8541.6743
EC00796=0.0000,8544.4402
EC00797=0.0000,8547.2469
EC00798=0.0000,8550.0000
EC00799=0.0000,8552.7531
EC00800=0.0000,8555.5598
EC00801=0.0000,8558.3257
EC00802=0.0000,8559.7254
EC00803=0.0000,8560.3637
EC00804=0.0000,8560.7187
EC00805=0.0000,8561.0200
EC00806=0.0000,8561.5211
EC00807=0.0000,8563.0317
EC00808=0.0000,8565.3479
EC00809=0.0000,8568.1086
EC00810=0.0000,8571.0234
EC00811=0.0000,8573.9765
EC00812=0.0000,8576.8914
EC00813=0.0000,8579.6519
EC00814=0.0000,8581.9680
EC00815=0.0000,8583.4791
EC00816=0.0000,8583.9803
EC00817=0.0000,8584.2813
EC00818=0.0000,8584.6359
EC00819=0.0000,8585.2745
EC00820=0.0000,8586.6744
EC00821=0.0000,8589.4401
EC00822=0.0000,8592.2471
EC00823=0.0000,8595.0000
EC00824=0.0000,8597.7529
EC00825=0.0000,8600.5599
EC00826=0.0000,8603.3256
EC00827=0.0000,8604.7255
EC00828=0.0000,8605.3641
EC00829=0.0000,8605.7187
EC00830=0.0000,8606.0197
EC00831=0.0000,8606.5209
EC00832=0.0000,8608.0320
EC00833=0.0000,8610.3481
EC00834=0.0000,8613.1086
EC00835=0.0000,8616.0235
EC00836=0.0000,8618.9766
EC00837=0.0000,8621.8914
EC00838=0.0000,8624.6521
EC00839=0.0000,8626.9683
EC00840=0.0000,8628.4789
EC00841=0.0000,8628.9800
EC00842=0.0000,8629.2813
EC00843=0.0000,8629.6363
EC00844=0.0000,8630.2746
EC00845=0.0000,8631.6743
EC00846=0.0000,8634.4402
EC00847=0.0000,8637.2469
EC00848=0.0000,8640.0000
EC00849=0.0000,8640.0000
EC00850=0.0000,8642.7075
EC00851=0.0000,8645.4993
EC00852=0.0000,8648.2758
EC00853=0.0000,8649.6431
EC00854=0.0000,8650.2359
EC00855=0.0000,8650.5465
EC00856=0.0000,8650.8039
EC00857=0.0000,8651.2607
EC00858=0.0000,8652.7735
EC00859=0.0000,8655.1340
EC00860=0.0000,8657.9686
EC00861=0.0000,8660.9753
EC00862=0.0000,8664.0247
EC00863=0.0000,8667.0314
EC00864=0.0000,8669.8659
EC00865=0.0000,8672.2261
EC00866=0.0000,8673.7397
EC00867=0.0000,8674.1962
EC00868=0.0000,8674.4534
EC00869=0.0000,8674.7640
EC00870=0.0000,8675.3567
EC00871=0.0000,8676.7241
EC00872=0.0000,8679.5007
EC00873=0.0000,8682.2930
EC00874=0.0000,8685.0000
EC00875=0.0000,8687.7070
EC00876=0.0000,8690.4999
EC00877=0.0000,8693.2759
EC00878=0.0000,8694.6433
EC00879=0.0000,8695.2360
EC00880=0.0000,8695.5466
EC00881=0.0000,8695.8038
EC00882=0.0000,8696.2603
EC00883=0.0000,8697.7739
EC00884=0.0000,8700.1341
EC00885=0.0000,8702.9686
EC00886=0.0000,8705.9753
EC00887=0.0000,8709.0247
EC00888=0.0000,8712.0314
EC00889=0.0000,8714.8660
EC00890=0.0000,8717.2265
EC00891=0.0000,8718.7393
EC00892=0.0000,8719.1961
EC00893=0.0000,8719.4535
EC00894=0.0000,8719.7641
EC00895=0.0000,8720.3569
EC00896=0.0000,8721.7242
EC00897=0.0000,8724.5007
EC00898=0.0000,8727.2925
EC00899=0.0000,8730.0000
EC00900=0.0000,8732.7075
EC00901=0.0000,8735.4993
EC00902=0.0000,8738.2758
EC00903=0.0000,8739.6431
EC00904=0.0000,8740.2359
EC00905=0.0000,8740.5465
EC00906=0.0000,8740.8039
EC00907=0.0000,8741.2607
EC00908=0.0000,8742.7735
EC00909=0.0000,8745.1340
EC00910=0.0000,8747.9686
EC00911=0.0000,8750.9753
EC00912=0.0000,8754.0247
EC00913=0.0000,8757.0314
EC00914=0.0000,8759.8659
EC00915=0.0000,8762.2261
EC00916=0.0000,8763.7397
EC00917=0.0000,8764.1962
EC00918=0.0000,8764.4534
EC00919=0.0000,8764.7640
EC00920=0.0000,8765.3567
EC00921=0.0000,8766.7241
EC00922=0.0000,8769.5007
EC00923=0.0000,8772.2930
EC00924=0.0000,8775.0000
EC00925=0.0000,8777.7070
EC00926=0.0000,8780.4999
EC00927=0.0000,8783.2759
EC00928=0.0000,8784.6433
EC00929=0.0000,8785.2360
EC00930=0.0000,8785.5466
EC00931=0.0000,8785.8038
EC00932=0.0000,8786.2603
EC00933=0.0000,8787.7739
EC00934=0.0000,8790.1341
EC00935=0.0000,8792.9686
EC00936=0.0000,8795.9753
EC00937=0.0000,8799.0247
EC00938=0.0000,8802.0314
EC00939=0.0000,8804.8660
EC00940=0.0000,8807.2265
EC00941=0.0000,8808.7393
EC00942=0.0000,8809.1961
EC00943=0.0000,8809.4535
EC00944=0.0000,8809.7641
EC00945=0.0000,8810.3569
EC00946=0.0000,8811.7242
EC00947=0.0000,8814.5007
EC00948=0.0000,8817.2925
EC00949=0.0000,8820.0000
EC00950=0.0000,8820.0000
EC00951=0.0000,8822.7075
EC00952=0.0000,8825.4993
EC00953=0.0000,8828.2758
EC00954=0.0000,8829.6431
EC00955=0.0000,8830.2359
EC00956=0.0000,8830.5465
EC00957=0.0000,8830.8039
EC00958=0.0000,8831.2607
EC00959=0.0000,8832.7735
EC00960=0.0000,8835.1340
EC00961=0.0000,8837.9686
EC00962=0.0000,8840.9753
EC00963=0.0000,8844.0247
EC00964=0.0000,8847.0314
EC00965=0.0000,8849.8659
EC00966=0.0000,8852.2261
EC00967=0.0000,8853.7397
EC00968=0.0000,8854.1962
EC00969=0.0000,8854.4534
EC00970=0.0000,8854.7640
EC00971=0.0000,8855.3567
EC00972=0.0000,8856.7241
EC00973=0.0000,8859.5007
EC00974=0.0000,8862.2930
EC00975=0.0000,8865.0000
EC00976=0.0000,8867.7070
EC00977=0.0000,8870.4999
EC00978=0.0000,8873.2759
EC00979=0.0000,8874.6433
EC00980=0.0000,8875.2360
EC00981=0.0000,8875.5466
EC00982=0.0000,8875.8038
EC00983=0.0000,8876.2603
EC00984=0.0000,8877.7739
EC00985=0.0000,8880.1341
EC00986=0.0000,8882.9686
EC00987=0.0000,8885.9753
EC00988=0.0000,8889.0247
EC00989=0.0000,8892.0314
EC00990=0.0000,8894.8660
EC00991=0.0000,8897.2265
EC00992=0.0000,8898.7393
EC00993=0.0000,8899.1961
EC00994=0.0000,8899.4535
EC00995=0.0000,8899.7641
EC00996=0.0000,8900.3569
EC00997=0.0000,8901.7242
EC00998=0.0000,8904.5007
EC00999=0.0000,8907.2925
EC01000=0.0000,8910.0000
EC01001=0.0000,8912.7075
EC01002=0.0000,8915.4993
EC01003=0.0000,8918.2758
EC01004=0.0000,8919.6431
EC01005=0.0000,8920.2359
EC01006=0.0000,8920.5465
EC01007=0.0000,8920.8039
EC01008=0.0000,8921.2607
EC01009=0.0000,8922.7735
EC01010=0.0000,8925.1340
EC01011=0.0000,8927.9686
EC01012=0.0000,8930.9753
EC01013=0.0000,8934.0247
EC01014=0.0000,8937.0314
EC01015=0.0000,8939.8659
EC01016=0.0000,8942.2261
EC01017=0.0000,8943.7397
EC01018=0.0000,8944.1962
EC01019=0.0000,8944.4534
EC01020=0.0000,8944.7640
EC01021=0.0000,8945.3567
EC01022=0.0000,8946.7241
EC01023=0.0000,8949.5007
EC01024=0.0000,8952.2930
EC01025=0.0000,8955.0000
EC01026=0.0000,8957.7070
EC01027=0.0000,8960.4999
EC01028=0.0000,8963.2759
EC01029=0.0000,8964.6433
EC01030=0.0000,8965.2360
EC01031=0.0000,8965.5466
EC01032=0.0000,8965.8038
EC01033=0.0000,8966.2603
EC01034=0.0000,8967.7739
EC01035=0.0000,8970.1341
EC01036=0.0000,8972.9686
EC01037=0.0000,8975.9753
EC01038=0.0000,8979.0247
EC01039=0.0000,8982.0314
EC01040=0.0000,8984.8660
EC01041=0.0000,8987.2265
EC01042=0.0000,8988.7393
EC01043=0.0000,8989.1961
EC01044=0.0000,8989.4535
EC01045=0.0000,8989.7641
EC01046=0.0000,8990.3569
EC01047=0.0000,8991.7242
EC01048=0.0000,8994.5007
EC01049=0.0000,8997.2925
EC01050=0.0000,9000.0000
EC01051=0.0000,9000.0000
EC01052=0.0000,9002.6603
EC01053=0.0000,9005.4368
EC01054=0.0000,9008.2235
EC01055=0.0000,9009.5577
EC01056=0.0000,9010.1045
EC01057=0.0000,9010.3719
EC01058=0.0000,9010.5864
EC01059=0.0000,9010.9998
EC01060=0.0000,9012.5167
EC01061=0.0000,9014.9212
EC01062=0.0000,9017.8298
EC01063=0.0000,9020.9268
EC01064=0.0000,9024.0730
EC01065=0.0000,9027.1707
EC01066=0.0000,9030.0788
EC01067=0.0000,9032.4830
EC01068=0.0000,9034.0000
EC01069=0.0000,9034.4140
EC01070=0.0000,9034.6279
EC01071=0.0000,9034.8952
EC01072=0.0000,9035.4421
EC01073=0.0000,9036.7764
EC01074=0.0000,9039.5628
EC01075=0.0000,9042.3404
EC01076=0.0000,9045.0000
EC01077=0.0000,9047.6596
EC01078=0.0000,9050.4372
EC01079=0.0000,9053.2236
EC01080=0.0000,9054.5579
EC01081=0.0000,9055.1048
EC01082=0.0000,9055.3721
EC01083=0.0000,9055.5860
EC01084=0.0000,9056.0000
EC01085=0.0000,9057.5170
EC01086=0.0000,9059.9212
EC01087=0.0000,9062.8293
EC01088=0.0000,9065.9270
EC01089=0.0000,9069.0732
EC01090=0.0000,9072.1702
EC01091=0.0000,9075.0788
EC01092=0.0000,9077.4833
EC01093=0.0000,9079.0002
EC01094=0.0000,9079.4136
EC01095=0.0000,9079.6281
EC01096=0.0000,9079.8955
EC01097=0.0000,9080.4423
EC01098=0.0000,9081.7765
EC01099=0.0000,9084.5632
EC01100=0.0000,9087.3397
EC01101=0.0000,9090.0000
EC01102=0.0000,9092.6603
EC01103=0.0000,9095.4368
EC01104=0.0000,9098.2235
EC01105=0.0000,9099.5577
EC01106=0.0000,9100.1045
EC01107=0.0000,9100.3719
EC01108=0.0000,9100.5864
EC01109=0.0000,9100.9998
EC01110=0.0000,9102.5167
EC01111=0.0000,9104.9212
EC01112=0.0000,9107.8298
EC01113=0.0000,9110.9268
EC01114=0.0000,9114.0730
EC01115=0.0000,9117.1707
EC01116=0.0000,9120.0788
EC01117=0.0000,9122.4830
EC01118=0.0000,9124.0000
EC01119=0.0000,9124.4140
EC01120=0.0000,9124.6279
EC01121=0.0000,9124.8952
EC01122=0.0000,9125.4421
EC01123=0.0000,9126.7764
EC01124=0.0000,9129.5628
EC01125=0.0000,9132.3404
EC01126=0.0000,9135.0000
EC01127=0.0000,9137.6596
EC01128=0.0000,9140.4372
EC01129=0.0000,9143.2236
EC01130=0.0000,9144.5579
EC01131=0.0000,9145.1048
EC01132=0.0000,9145.3721
EC01133=0.0000,9145.5860
EC01134=0.0000,9146.0000
EC01135=0.0000,9147.5170
EC01136=0.0000,9149.9212
EC01137=0.0000,9152.8293
EC01138=0.0000,9155.9270
EC01139=0.0000,9159.0732
EC01140=0.0000,9162.1702
EC01141=0.0000,9165.0788
EC01142=0.0000,9167.4833
EC01143=0.0000,9169.0002
EC01144=0.0000,9169.4136
EC01145=0.0000,9169.6281
EC01146=0.0000,9169.8955
EC01147=0.0000,9170.4423
EC01148=0.0000,9171.7765
EC01149=0.0000,9174.5632
EC01150=0.0000,9177.3397
EC01151=0.0000,9180.0000
EC01152=0.0000,9180.0000
EC01153=0.0000,9182.6603
EC01154=0.0000,9185.4368
EC01155=0.0000,9188.2235
EC01156=0.0000,9189.5577
EC01157=0.0000,9190.1045
EC01158=0.0000,9190.3719
EC01159=0.0000,9190.5864
EC01160=0.0000,9190.9998
EC01161=0.0000,9192.5167
EC01162=0.0000,9194.9212
EC01163=0.0000,9197.8298
EC01164=0.0000,9200.9268
EC01165=0.0000,9204.0730
EC01166=0.0000,9207.1707
EC01167=0.0000,9210.0788
EC01168=0.0000,9212.4830
EC01169=0.0000,9214.0000
EC01170=0.0000,9214.4140
EC01171=0.0000,9214.6279
EC01172=0.0000,9214.8952
EC01173=0.0000,9215.4421
EC01174=0.0000,9216.7764
EC01175=0.0000,9219.5628
EC01176=0.0000,9222.3404
EC01177=0.0000,9225.0000
EC01178=0.0000,9227.6596
EC01179=0.0000,9230.4372
EC01180=0.0000,9233.2236
EC01181=0.0000,9234.5579
EC01182=0.0000,9235.1048
EC01183=0.0000,9235.3721
EC01184=0.0000,9235.5860
EC01185=0.0000,9236.0000
EC01186=0.0000,9237.5170
EC01187=0.0000,9239.9212
EC01188=0.0000,9242.8293
EC01189=0.0000,9245.9270
EC01190=0.0000,9249.0732
EC01191=0.0000,9252.1702
EC01192=0.0000,9255.0788
EC01193=0.0000,9257.4833
EC01194=0.0000,9259.0002
EC01195=0.0000,9259.4136
EC01196=0.0000,9259.6281
EC01197=0.0000,9259.8955
EC01198=0.0000,9260.4423
EC01199=0.0000,9261.7765
EC01200=0.0000,9264.5632
EC01201=0.0000,9267.3397
EC01202=0.0000,9270.0000
EC01203=0.0000,9272.6603
EC01204=0.0000,9275.4368
EC01205=0.0000,9278.2235
EC01206=0.0000,9279.5577
EC01207=0.0000,9280.1045
EC01208=0.0000,9280.3719
EC01209=0.0000,9280.5864
EC01210=0.0000,9280.9998
EC01211=0.0000,9282.5167
EC01212=0.0000,9284.9212
EC01213=0.0000,9287.8298
EC01214=0.0000,9290.9268
EC01215=0.0000,9294.0730
EC01216=0.0000,9297.1707
EC01217=0.0000,9300.0788
EC01218=0.0000,9302.4830
EC01219=0.0000,9304.0000
EC01220=0.0000,9304.4140
EC01221=0.0000,9304.6279
EC01222=0.0000,9304.8952
EC01223=0.0000,9305.4421
EC01224=0.0000,9306.7764
EC01225=0.0000,9309.5628
EC01226=0.0000,9312.3404
EC01227=0.0000,9315.0000
EC01228=0.0000,9317.6596
EC01229=0.0000,9320.4372
EC01230=0.0000,9323.2236
EC01231=0.0000,9324.5579
EC01232=0.0000,9325.1048
EC01233=0.0000,9325.3721
EC01234=0.0000,9325.5860
EC01235=0.0000,9326.0000
EC01236=0.0000,9327.5170
EC01237=0.0000,9329.9212
EC01238=0.0000,9332.8293
EC01239=0.0000,9335.9270
EC01240=0.0000,9339.0732
EC01241=0.0000,9342.1702
EC01242=0.0000,9345.0788
EC01243=0.0000,9347.4833
EC01244=0.0000,9349.0002
EC01245=0.0000,9349.4136
EC01246=0.0000,9349.6281
EC01247=0.0000,9349.8955
EC01248=0.0000,9350.4423
EC01249=0.0000,9351.7765
EC01250=0.0000,9354.5632
EC01251=0.0000,9357.3397
EC01252=0.0000,9360.0000
EC01253=0.0000,9360.0000
EC01254=0.0000,9362.6105
EC01255=0.0000,9365.3720
EC01256=0.0000,9368.1701
EC01257=0.0000,9369.4699
EC01258=0.0000,9369.9705
EC01259=0.0000,9370.1944
EC01260=0.0000,9370.3679
EC01261=0.0000,9370.7398
EC01262=0.0000,9372.2618
EC01263=0.0000,9374.7112
EC01264=0.0000,9377.6927
EC01265=0.0000,9380.8797
EC01266=0.0000,9384.1202
EC01267=0.0000,9387.3076
EC01268=0.0000,9390.2891
EC01269=0.0000,9392.7379
EC01270=0.0000,9394.2600
EC01271=0.0000,9394.6321
EC01272=0.0000,9394.8056
EC01273=0.0000,9395.0300
EC01274=0.0000,9395.5299
EC01275=0.0000,9396.8301
EC01276=0.0000,9399.6279
EC01277=0.0000,9402.3891
EC01278=0.0000,9405.0000
EC01279=0.0000,9407.6109
EC01280=0.0000,9410.3721
EC01281=0.0000,9413.1699
EC01282=0.0000,9414.4701
EC01283=0.0000,9414.9700
EC01284=0.0000,9415.1944
EC01285=0.0000,9415.3679
EC01286=0.0000,9415.7400
EC01287=0.0000,9417.2621
EC01288=0.0000,9419.7109
EC01289=0.0000,9422.6924
EC01290=0.0000,9425.8798
EC01291=0.0000,9429.1203
EC01292=0.0000,9432.3073
EC01293=0.0000,9435.2888
EC01294=0.0000,9437.7382
EC01295=0.0000,9439.2602
EC01296=0.0000,9439.6321
EC01297=0.0000,9439.8056
EC01298=0.0000,9440.0295
EC01299=0.0000,9440.5301
EC01300=0.0000,9441.8299
EC01301=0.0000,9444.6280
EC01302=0.0000,9447.3895
EC01303=0.0000,9450.0000
EC01304=0.0000,9452.6105
EC01305=0.0000,9455.3720
EC01306=0.0000,9458.1701
EC01307=0.0000,9459.4699
EC01308=0.0000,9459.9705
EC01309=0.0000,9460.1944
EC01310=0.0000,9460.3679
EC01311=0.0000,9460.7398
EC01312=0.0000,9462.2618
EC01313=0.0000,9464.7112
EC01314=0.0000,9467.6927
EC01315=0.0000,9470.8797
EC01316=0.0000,9474.1202
EC01317=0.0000,9477.3076
EC01318=0.0000,9480.2891
EC01319=0.0000,9482.7379
EC01320=0.0000,9484.2600
EC01321=0.0000,9484.6321
EC01322=0.0000,9484.8056
EC01323=0.0000,9485.0300
EC01324=0.0000,9485.5299
EC01325=0.0000,9486.8301
EC01326=0.0000,9489.6279
EC01327=0.0000,9492.3891
EC01328=0.0000,9495.0000
EC01329=0.0000,9497.6109
EC01330=0.0000,9500.3721
EC01331=0.0000,9503.1699
EC01332=0.0000,9504.4701
EC01333=0.0000,9504.9700
EC01334=0.0000,9505.1944
EC01335=0.0000,9505.3679
EC01336=0.0000,9505.7400
EC01337=0.0000,9507.2621
EC01338=0.0000,9509.7109
EC01339=0.0000,9512.6924
EC01340=0.0000,9515.8798
EC01341=0.0000,9519.1203
EC01342=0.0000,9522.3073
EC01343=0.0000,9525.2888
EC01344=0.0000,9527.7382
EC01345=0.0000,9529.2602
EC01346=0.0000,9529.6321
EC01347=0.0000,9529.8056
EC01348=0.0000,9530.0295
EC01349=0.0000,9530.5301
EC01350=0.0000,9531.8299
EC01351=0.0000,9534.6280
EC01352=0.0000,9537.3895
EC01353=0.0000,9540.0000
EC01354=0.0000,9540.0000
EC01355=0.0000,9542.6105
EC01356=0.0000,9545.3720
EC01357=0.0000,9548.1701
EC01358=0.0000,9549.4699
EC01359=0.0000,9549.9705
EC01360=0.0000,9550.1944
EC01361=0.0000,9550.3679
EC01362=0.0000,9550.7398
EC01363=0.0000,9552.2618
EC01364=0.0000,9554.7112
EC01365=0.0000,9557.6927
EC01366=0.0000,9560.8797
EC01367=0.0000,9564.1202
EC01368=0.0000,9567.3076
EC01369=0.0000,9570.2891
EC01370=0.0000,9572.7379
EC01371=0.0000,9574.2600
EC01372=0.0000,9574.6321
EC01373=0.0000,9574.8056
EC01374=0.0000,9575.0300
EC01375=0.0000,9575.5299
EC01376=0.0000,9576.8301
EC01377=0.0000,9579.6279
EC01378=0.0000,9582.3891
EC01379=0.0000,9585.0000
EC01380=0.0000,9587.6109
EC01381=0.0000,9590.3721
EC01382=0.0000,9593.1699
EC01383=0.0000,9594.4701
EC01384=0.0000,9594.9700
EC01385=0.0000,9595.1944
EC01386=0.0000,9595.3679
EC01387=0.0000,9595.7400
EC01388=0.0000,9597.2621
EC01389=0.0000,9599.7109
EC01390=0.0000,9602.6924
EC01391=0.0000,9605.8798
EC01392=0.0000,9609.1203
EC01393=0.0000,9612.3073
EC01394=0.0000,9615.2888
EC01395=0.0000,9617.7382
EC01396=0.0000,9619.2602
EC01397=0.0000,9619.6321
EC01398=0.0000,9619.8056
EC01399=0.0000,9620.0295
EC01400=0.0000,9620.5301
EC01401=0.0000,9621.8299
EC01402=0.0000,9624.6280
EC01403=0.0000,9627.3895
EC01404=0.0000,9630.0000
EC01405=0.0000,9632.6105
EC01406=0.0000,9635.3720
EC01407=0.0000,9638.1701
EC01408=0.0000,9639.4699
EC01409=0.0000,9639.9705
EC01410=0.0000,9640.1944
EC01411=0.0000,9640.3679
EC01412=0.0000,9640.7398
EC01413=0.0000,9642.2618
EC01414=0.0000,9644.7112
EC01415=0.0000,9647.6927
EC01416=0.0000,9650.8797
EC01417=0.0000,9654.1202
EC01418=0.0000,9657.3076
EC01419=0.0000,9660.2891
EC01420=0.0000,9662.7379
EC01421=0.0000,9664.2600
EC01422=0.0000,9664.6321
EC01423=0.0000,9664.8056
EC01424=0.0000,9665.0300
EC01425=0.0000,9665.5299
EC01426=0.0000,9666.8301
EC01427=0.0000,9669.6279
EC01428=0.0000,9672.3891
EC01429=0.0000,9675.0000
EC01430=0.0000,9677.6109
EC01431=0.0000,9680.3721
EC01432=0.0000,9683.1699
EC01433=0.0000,9684.4701
EC01434=0.0000,9684.9700
EC01435=0.0000,9685.1944
EC01436=0.0000,9685.3679
EC01437=0.0000,9685.7400
EC01438=0.0000,9687.2621
EC01439=0.0000,9689.7109
EC01440=0.0000,9692.6924
EC01441=0.0000,9695.8798
EC01442=0.0000,9699.1203
EC01443=0.0000,9702.3073
EC01444=0.0000,9705.2888
EC01445=0.0000,9707.7382
EC01446=0.0000,9709.2602
EC01447=0.0000,9709.6321
EC01448=0.0000,9709.8056
EC01449=0.0000,9710.0295
EC01450=0.0000,9710.5301
EC01451=0.0000,9711.8299
EC01452=0.0000,9714.6280
EC01453=0.0000,9717.3895
EC01454=0.0000,9720.0000
EC01455=0.0000,9720.0000
EC01456=0.0000,9722.5595
EC01457=0.0000,9725.3045
EC01458=0.0000,9728.1135
EC01459=0.0000,9729.3788
EC01460=0.0000,9729.8327
EC01461=0.0000,9730.0151
EC01462=0.0000,9730.1489
EC01463=0.0000,9730.4816
EC01464=0.0000,9732.0102
EC01465=0.0000,9734.5040
EC01466=0.0000,9737.5575
EC01467=0.0000,9740.8329
EC01468=0.0000,9744.1669
EC01469=0.0000,9747.4422
EC01470=0.0000,9750.4960
EC01471=0.0000,9752.9901
EC01472=0.0000,9754.5184
EC01473=0.0000,9754.8513
EC01474=0.0000,9754.9851
EC01475=0.0000,9755.1672
EC01476=0.0000,9755.6212
EC01477=0.0000,9756.8860
EC01478=0.0000,9759.6950
EC01479=0.0000,9762.4397
EC01480=0.0000,9765.0000
EC01481=0.0000,9767.5591
EC01482=0.0000,9770.3050
EC01483=0.0000,9773.1140
EC01484=0.0000,9774.3788
EC01485=0.0000,9774.8328
EC01486=0.0000,9775.0149
EC01487=0.0000,9775.1487
EC01488=0.0000,9775.4816
EC01489=0.0000,9777.0099
EC01490=0.0000,9779.5040
EC01491=0.0000,9782.5578
EC01492=0.0000,9785.8331
EC01493=0.0000,9789.1671
EC01494=0.0000,9792.4425
EC01495=0.0000,9795.4960
EC01496=0.0000,9797.9898
EC01497=0.0000,9799.5184
EC01498=0.0000,9799.8511
EC01499=0.0000,9799.9849
EC01500=0.0000,9800.1673
EC01501=0.0000,9800.6212
EC01502=0.0000,9801.8865
EC01503=0.0000,9804.6955
EC01504=0.0000,9807.4405
EC01505=0.0000,9810.0000
EC01506=0.0000,9812.5595
EC01507=0.0000,9815.3053
EC01508=0.0000,9818.1143
EC01509=0.0000,9819.3788
EC01510=0.0000,9819.8327
EC01511=0.0000,9820.0151
EC01512=0.0000,9820.1489
EC01513=0.0000,9820.4816
EC01514=0.0000,9822.0102
EC01515=0.0000,9824.5040
EC01516=0.0000,9827.5575
EC01517=0.0000,9830.8329
EC01518=0.0000,9834.1669
EC01519=0.0000,9837.4422
EC01520=0.0000,9840.4960
EC01521=0.0000,9842.9901
EC01522=0.0000,9844.5184
EC01523=0.0000,9844.8513
EC01524=0.0000,9844.9851
EC01525=0.0000,9845.1672
EC01526=0.0000,9845.6212
EC01527=0.0000,9846.8860
EC01528=0.0000,9849.6950
EC01529=0.0000,9852.4397
EC01530=0.0000,9855.0000
EC01531=0.0000,9857.5591
EC01532=0.0000,9860.3050
EC01533=0.0000,9863.1140
EC01534=0.0000,9864.3788
EC01535=0.0000,9864.8328
EC01536=0.0000,9865.0149
EC01537=0.0000,9865.1487
EC01538=0.0000,9865.4816
EC01539=0.0000,9867.0099
EC01540=0.0000,9869.5040
EC01541=0.0000,9872.5578
EC01542=0.0000,9875.8331
EC01543=0.0000,9879.1671
EC01544=0.0000,9882.4425
EC01545=0.0000,9885.4960
EC01546=0.0000,9887.9898
EC01547=0.0000,9889.5184
EC01548=0.0000,9889.8511
EC01549=0.0000,9889.9849
EC01550=0.0000,9890.1673
EC01551=0.0000,9890.6212
EC01552=0.0000,9891.8865
EC01553=0.0000,9894.6955
EC01554=0.0000,9897.4405
EC01555=0.0000,9900.0000
EC01556=0.0000,9900.0000
EC01557=0.0000,9902.5595
EC01558=0.0000,9905.3053
EC01559=0.0000,9908.1143
EC01560=0.0000,9909.3788
EC01561=0.0000,9909.8327
EC01562=0.0000,9910.0151
EC01563=0.0000,9910.1489
EC01564=0.0000,9910.4816
EC01565=0.0000,9912.0102
EC01566=0.0000,9914.5040
EC01567=0.0000,9917.5575
EC01568=0.0000,9920.8329
EC01569=0.0000,9924.1669
EC01570=0.0000,9927.4422
EC01571=0.0000,9930.4960
EC01572=0.0000,9932.9901
EC01573=0.0000,9934.5184
EC01574=0.0000,9934.8513
EC01575=0.0000,9934.9851
EC01576=0.0000,9935.1672
EC01577=0.0000,9935.6212
EC01578=0.0000,9936.8860
EC01579=0.0000,9939.6950
EC01580=0.0000,9942.4397
EC01581=0.0000,9945.0000
EC01582=0.0000,9947.5591
EC01583=0.0000,9950.3050
EC01584=0.0000,9953.1140
EC01585=0.0000,9954.3788
EC01586=0.0000,9954.8328
EC01587=0.0000,9955.0149
EC01588=0.0000,9955.1487
EC01589=0.0000,9955.4816
EC01590=0.0000,9957.0099
EC01591=0.0000,9959.5040
EC01592=0.0000,9962.5578
EC01593=0.0000,9965.8331
EC01594=0.0000,9969.1671
EC01595=0.0000,9972.4425
EC01596=0.0000,9975.4960
EC01597=0.0000,9977.9898
EC01598=0.0000,9979.5184
EC01599=0.0000,9979.8511
EC01600=0.0000,9979.9849
EC01601=0.0000,9980.1673
EC01602=0.0000,9980.6212
EC01603=0.0000,9981.8865
EC01604=0.0000,9984.6955
EC01605=0.0000,9987.4405
EC01606=0.0000,9990.0000
EC01607=0.0000,9992.5595
EC01608=0.0000,9995.3053
EC01609=0.0000,9998.1143
EC01610=0.0000,9999.3788
EC01611=0.0000,9999.8327
EC01612=0.0000,10000.0151
EC01613=0.0000,10000.1489
EC01614=0.0000,10000.4816
EC01615=0.0000,10002.0102
EC01616=0.0000,10004.5040
EC01617=0.0000,10007.5575
EC01618=0.0000,10010.8329
EC01619=0.0000,10014.1669
EC01620=0.0000,10017.4422
EC01621=0.0000,10020.4960
EC01622=0.0000,10022.9901
EC01623=0.0000,10024.5184
EC01624=0.0000,10024.8513
EC01625=0.0000,10024.9851
EC01626=0.0000,10025.1672
EC01627=0.0000,10025.6212
EC01628=0.0000,10026.8860
EC01629=0.0000,10029.6950
EC01630=0.0000,10032.4397
EC01631=0.0000,10035.0000
EC01632=0.0000,10037.5591
EC01633=0.0000,10040.3050
EC01634=0.0000,10043.1140
EC01635=0.0000,10044.3788
EC01636=0.0000,10044.8328
EC01637=0.0000,10045.0149
EC01638=0.0000,10045.1487
EC01639=0.0000,10045.4816
EC01640=0.0000,10047.0099
EC01641=0.0000,10049.5040
EC01642=0.0000,10052.5578
EC01643=0.0000,10055.8331
EC01644=0.0000,10059.1671
EC01645=0.0000,10062.4425
EC01646=0.0000,10065.4960
EC01647=0.0000,10067.9898
EC01648=0.0000,10069.5184
EC01649=0.0000,10069.8511
EC01650=0.0000,10069.9849
EC01651=0.0000,10070.1673
EC01652=0.0000,10070.6212
EC01653=0.0000,10071.8857
EC01654=0.0000,10074.6947
EC01655=0.0000,10077.4405
EC01656=0.0000,10080.0000
EC01657=0.0000,10080.0000
EC01658=0.0000,10082.5072
EC01659=0.0000,10085.2349
EC01660=0.0000,10088.0561
EC01661=0.0000,10089.2852
EC01662=0.0000,10089.6930
EC01663=0.0000,10089.8344
EC01664=0.0000,10089.9312
EC01665=0.0000,10090.2265
EC01666=0.0000,10091.7624
EC01667=0.0000,10094.3014
EC01668=0.0000,10097.4259
EC01669=0.0000,10100.7876
EC01670=0.0000,10104.2123
EC01671=0.0000,10107.5744
EC01672=0.0000,10110.6985
EC01673=0.0000,10113.2374
EC01674=0.0000,10114.7737
EC01675=0.0000,10115.0694
EC01676=0.0000,10115.1660
EC01677=0.0000,10115.3073
EC01678=0.0000,10115.7148
EC01679=0.0000,10116.9441
EC01680=0.0000,10119.7651
EC01681=0.0000,10122.4931
EC01682=0.0000,10125.0000
EC01683=0.0000,10127.5069
EC01684=0.0000,10130.2349
EC01685=0.0000,10133.0566
EC01686=0.0000,10134.2852
EC01687=0.0000,10134.6927
EC01688=0.0000,10134.8340
EC01689=0.0000,10134.9306
EC01690=0.0000,10135.2263
EC01691=0.0000,10136.7626
EC01692=0.0000,10139.3015
EC01693=0.0000,10142.4256
EC01694=0.0000,10145.7877
EC01695=0.0000,10149.2124
EC01696=0.0000,10152.5741
EC01697=0.0000,10155.6986
EC01698=0.0000,10158.2376
EC01699=0.0000,10159.7735
EC01700=0.0000,10160.0688
EC01701=0.0000,10160.1656
EC01702=0.0000,10160.3070
EC01703=0.0000,10160.7148
EC01704=0.0000,10161.9439
EC01705=0.0000,10164.7651
EC01706=0.0000,10167.4928
EC01707=0.0000,10170.0000
EC01708=0.0000,10172.5064
EC01709=0.0000,10175.2349
EC01710=0.0000,10178.0561
EC01711=0.0000,10179.2852
EC01712=0.0000,10179.6930
EC01713=0.0000,10179.8344
EC01714=0.0000,10179.9312
EC01715=0.0000,10180.2265
EC01716=0.0000,10181.7624
EC01717=0.0000,10184.3014
EC01718=0.0000,10187.4259
EC01719=0.0000,10190.7876
EC01720=0.0000,10194.2123
EC01721=0.0000,10197.5744
EC01722=0.0000,10200.6985
EC01723=0.0000,10203.2374
EC01724=0.0000,10204.7737
EC01725=0.0000,10205.0694
EC01726=0.0000,10205.1660
EC01727=0.0000,10205.3073
EC01728=0.0000,10205.7148
EC01729=0.0000,10206.9441
EC01730=0.0000,10209.7651
EC01731=0.0000,10212.4931
EC01732=0.0000,10215.0000
EC01733=0.0000,10217.5069
EC01734=0.0000,10220.2349
EC01735=0.0000,10223.0566
EC01736=0.0000,10224.2852
EC01737=0.0000,10224.6927
EC01738=0.0000,10224.8340
EC01739=0.0000,10224.9306
EC01740=0.0000,10225.2263
EC01741=0.0000,10226.7626
EC01742=0.0000,10229.3015
EC01743=0.0000,10232.4256
EC01744=0.0000,10235.7877
EC01745=0.0000,10239.2124
EC01746=0.0000,10242.5741
EC01747=0.0000,10245.6986
EC01748=0.0000,10248.2376
EC01749=0.0000,10249.7735
EC01750=0.0000,10250.0688
EC01751=0.0000,10250.1656
EC01752=0.0000,10250.3070
EC01753=0.0000,10250.7148
EC01754=0.0000,10251.9439
EC01755=0.0000,10254.7651
EC01756=0.0000,10257.4928
EC01757=0.0000,10260.0000
EC01758=0.0000,10260.0000
EC01759=0.0000,10262.5064
EC01760=0.0000,10265.2349
EC01761=0.0000,10268.0561
EC01762=0.0000,10269.2852
EC01763=0.0000,10269.6930
EC01764=0.0000,10269.8344
EC01765=0.0000,10269.9312
EC01766=0.0000,10270.2265
EC01767=0.0000,10271.7624
EC01768=0.0000,10274.3014
EC01769=0.0000,10277.4259
EC01770=0.0000,10280.7876
EC01771=0.0000,10284.2123
EC01772=0.0000,10287.5744
EC01773=0.0000,10290.6985
EC01774=0.0000,10293.2374
EC01775=0.0000,10294.7737
EC01776=0.0000,10295.0694
EC01777=0.0000,10295.1660
EC01778=0.0000,10295.3073
EC01779=0.0000,10295.7148
EC01780=0.0000,10296.9441
EC01781=0.0000,10299.7651
EC01782=0.0000,10302.4931
EC01783=0.0000,10305.0000
EC01784=0.0000,10307.5069
EC01785=0.0000,10310.2349
EC01786=0.0000,10313.0566
EC01787=0.0000,10314.2852
EC01788=0.0000,10314.6927
EC01789=0.0000,10314.8340
EC01790=0.0000,10314.9306
EC01791=0.0000,10315.2263
EC01792=0.0000,10316.7626
EC01793=0.0000,10319.3015
EC01794=0.0000,10322.4256
EC01795=0.0000,10325.7877
EC01796=0.0000,10329.2124
EC01797=0.0000,10332.5741
EC01798=0.0000,10335.6986
EC01799=0.0000,10338.2376
EC01800=0.0000,10339.7735
EC01801=0.0000,10340.0688
EC01802=0.0000,10340.1656
EC01803=0.0000,10340.3070
EC01804=0.0000,10340.7148
EC01805=0.0000,10341.9439
EC01806=0.0000,10344.7651
EC01807=0.0000,10347.4928
EC01808=0.0000,10350.0000
EC01809=0.0000,10352.5064
EC01810=0.0000,10355.2349
EC01811=0.0000,10358.0561
EC01812=0.0000,10359.2852
EC01813=0.0000,10359.6930
EC01814=0.0000,10359.8344
EC01815=0.0000,10359.9312
EC01816=0.0000,10360.2265
EC01817=0.0000,10361.7624
EC01818=0.0000,10364.3014
EC01819=0.0000,10367.4259
EC01820=0.0000,10370.7876
EC01821=0.0000,10374.2123
EC01822=0.0000,10377.5744
EC01823=0.0000,10380.6985
EC01824=0.0000,10383.2374
EC01825=0.0000,10384.7737
EC01826=0.0000,10385.0694
EC01827=0.0000,10385.1660
EC01828=0.0000,10385.3073
EC01829=0.0000,10385.7148
EC01830=0.0000,10386.9441
EC01831=0.0000,10389.7651
EC01832=0.0000,10392.4931
EC01833=0.0000,10395.0000
EC01834=0.0000,10397.5069
EC01835=0.0000,10400.2349
EC01836=0.0000,10403.0566
EC01837=0.0000,10404.2852
EC01838=0.0000,10404.6927
EC01839=0.0000,10404.8340
EC01840=0.0000,10404.9306
EC01841=0.0000,10405.2263
EC01842=0.0000,10406.7626
EC01843=0.0000,10409.3015
EC01844=0.0000,10412.4256
EC01845=0.0000,10415.7877
EC01846=0.0000,10419.2124
EC01847=0.0000,10422.5741
EC01848=0.0000,10425.6986
EC01849=0.0000,10428.2376
EC01850=0.0000,10429.7735
EC01851=0.0000,10430.0688
EC01852=0.0000,10430.1656
EC01853=0.0000,10430.3070
EC01854=0.0000,10430.7148
EC01855=0.0000,10431.9439
EC01856=0.0000,10434.7651
EC01857=0.0000,10437.4936
EC01858=0.0000,10440.0000
EC01859=0.0000,10440.0000
EC01860=0.0000,10442.4517
EC01861=0.0000,10445.1629
EC01862=0.0000,10447.9963
EC01863=0.0000,10449.1897
EC01864=0.0000,10449.5501
EC01865=0.0000,10449.6525
EC01866=0.0000,10449.7146
EC01867=0.0000,10449.9757
EC01868=0.0000,10451.5206
EC01869=0.0000,10454.1038
EC01870=0.0000,10457.2974
EC01871=0.0000,10460.7433
EC01872=0.0000,10464.2566
EC01873=0.0000,10467.7026
EC01874=0.0000,10470.8962
EC01875=0.0000,10473.4793
EC01876=0.0000,10475.0245
EC01877=0.0000,10475.2855
EC01878=0.0000,10475.3476
EC01879=0.0000,10475.4495
EC01880=0.0000,10475.8105
EC01881=0.0000,10477.0038
EC01882=0.0000,10479.8372
EC01883=0.0000,10482.5482
EC01884=0.0000,10485.0000
EC01885=0.0000,10487.4518
EC01886=0.0000,10490.1628
EC01887=0.0000,10492.9966
EC01888=0.0000,10494.1895
EC01889=0.0000,10494.5505
EC01890=0.0000,10494.6524
EC01891=0.0000,10494.7145
EC01892=0.0000,10494.9755
EC01893=0.0000,10496.5207
EC01894=0.0000,10499.1038
EC01895=0.0000,10502.2974
EC01896=0.0000,10505.7434
EC01897=0.0000,10509.2567
EC01898=0.0000,10512.7026
EC01899=0.0000,10515.8962
EC01900=0.0000,10518.4794
EC01901=0.0000,10520.0243
EC01902=0.0000,10520.2854
EC01903=0.0000,10520.3475
EC01904=0.0000,10520.4499
EC01905=0.0000,10520.8103
EC01906=0.0000,10522.0037
EC01907=0.0000,10524.8371
EC01908=0.0000,10527.5483
EC01909=0.0000,10530.0000
EC01910=0.0000,10532.4517
EC01911=0.0000,10535.1629
EC01912=0.0000,10537.9963
EC01913=0.0000,10539.1897
EC01914=0.0000,10539.5501
EC01915=0.0000,10539.6525
EC01916=0.0000,10539.7146
EC01917=0.0000,10539.9757
EC01918=0.0000,10541.5206
EC01919=0.0000,10544.1038
EC01920=0.0000,10547.2974
EC01921=0.0000,10550.7433
EC01922=0.0000,10554.2566
EC01923=0.0000,10557.7026
EC01924=0.0000,10560.8962
EC01925=0.0000,10563.4793
EC01926=0.0000,10565.0245
EC01927=0.0000,10565.2855
EC01928=0.0000,10565.3476
EC01929=0.0000,10565.4495
EC01930=0.0000,10565.8105
EC01931=0.0000,10567.0038
EC01932=0.0000,10569.8372
EC01933=0.0000,10572.5482
EC01934=0.0000,10575.0000
EC01935=0.0000,10577.4518
EC01936=0.0000,10580.1628
EC01937=0.0000,10582.9966
EC01938=0.0000,10584.1895
EC01939=0.0000,10584.5505
EC01940=0.0000,10584.6524
EC01941=0.0000,10584.7145
EC01942=0.0000,10584.9755
EC01943=0.0000,10586.5207
EC01944=0.0000,10589.1038
EC01945=0.0000,10592.2974
EC01946=0.0000,10595.7434
EC01947=0.0000,10599.2567
EC01948=0.0000,10602.7026
EC01949=0.0000,10605.8962
EC01950=0.0000,10608.4794
EC01951=0.0000,10610.0243
EC01952=0.0000,10610.2854
EC01953=0.0000,10610.3475
EC01954=0.0000,10610.4499
EC01955=0.0000,10610.8103
EC01956=0.0000,10612.0037
EC01957=0.0000,10614.8371
EC01958=0.0000,10617.5483
EC01959=0.0000,10620.0000
EC01960=0.0000,10620.0000
EC01961=0.0000,10622.4517
EC01962=0.0000,10625.1629
EC01963=0.0000,10627.9963
EC01964=0.0000,10629.1897
EC01965=0.0000,10629.5501
EC01966=0.0000,10629.6525
EC01967=0.0000,10629.7146
EC01968=0.0000,10629.9757
EC01969=0.0000,10631.5206
EC01970=0.0000,10634.1038
EC01971=0.0000,10637.2974
EC01972=0.0000,10640.7433
EC01973=0.0000,10644.2566
EC01974=0.0000,10647.7026
EC01975=0.0000,10650.8962
EC01976=0.0000,10653.4793
EC01977=0.0000,10655.0245
EC01978=0.0000,10655.2855
EC01979=0.0000,10655.3476
EC01980=0.0000,10655.4495
EC01981=0.0000,10655.8105
EC01982=0.0000,10657.0038
EC01983=0.0000,10659.8372
EC01984=0.0000,10662.5482
EC01985=0.0000,10665.0000
EC01986=0.0000,10667.4518
EC01987=0.0000,10670.1628
EC01988=0.0000,10672.9966
EC01989=0.0000,10674.1895
EC01990=0.0000,10674.5505
EC01991=0.0000,10674.6524
EC01992=0.0000,10674.7145
EC01993=0.0000,10674.9755
EC01994=0.0000,10676.5207
EC01995=0.0000,10679.1038
EC01996=0.0000,10682.2974
EC01997=0.0000,10685.7434
EC01998=0.0000,10689.2567
EC01999=0.0000,10692.7026
//INST
///DATE 2021/02/10 13:51
///COMM
///ATTR SC,RW,RJ
////FRAME USER 2
///GROUP1 RB1
///GROUP2 ST1
NOP
SMOVL C00000 +MOVJ EC00000
SMOVL C00001 +MOVJ EC00001
SMOVL C00002 +MOVJ EC00002
SMOVL C00003 +MOVJ EC00003
SMOVL C00004 +MOVJ EC00004
SMOVL C00005 +MOVJ EC00005
SMOVL C00006 +MOVJ EC00006
SMOVL C00007 +MOVJ EC00007
SMOVL C00008 +MOVJ EC00008
SMOVL C00009 +MOVJ EC00009
SMOVL C00010 +MOVJ EC00010
SMOVL C00011 +MOVJ EC00011
SMOVL C00012 +MOVJ EC00012
SMOVL C00013 +MOVJ EC00013
SMOVL C00014 +MOVJ EC00014
SMOVL C00015 +MOVJ EC00015
SMOVL C00016 +MOVJ EC00016
SMOVL C00017 +MOVJ EC00017
SMOVL C00018 +MOVJ EC00018
SMOVL C00019 +MOVJ EC00019
SMOVL C00020 +MOVJ EC00020
SMOVL C00021 +MOVJ EC00021
SMOVL C00022 +MOVJ EC00022
SMOVL C00023 +MOVJ EC00023
SMOVL C00024 +MOVJ EC00024
SMOVL C00025 +MOVJ EC00025
SMOVL C00026 +MOVJ EC00026
SMOVL C00027 +MOVJ EC00027
SMOVL C00028 +MOVJ EC00028
SMOVL C00029 +MOVJ EC00029
SMOVL C00030 +MOVJ EC00030
SMOVL C00031 +MOVJ EC00031
SMOVL C00032 +MOVJ EC00032
SMOVL C00033 +MOVJ EC00033
SMOVL C00034 +MOVJ EC00034
SMOVL C00035 +MOVJ EC00035
SMOVL C00036 +MOVJ EC00036
SMOVL C00037 +MOVJ EC00037
SMOVL C00038 +MOVJ EC00038
SMOVL C00039 +MOVJ EC00039
SMOVL C00040 +MOVJ EC00040
SMOVL C00041 +MOVJ EC00041
SMOVL C00042 +MOVJ EC00042
SMOVL C00043 +MOVJ EC00043
SMOVL C00044 +MOVJ EC00044
SMOVL C00045 +MOVJ EC00045
SMOVL C00046 +MOVJ EC00046
SMOVL C00047 +MOVJ EC00047
SMOVL C00048 +MOVJ EC00048
SMOVL C00049 +MOVJ EC00049
SMOVL C00050 +MOVJ EC00050
SMOVL C00051 +MOVJ EC00051
SMOVL C00052 +MOVJ EC00052
SMOVL C00053 +MOVJ EC00053
SMOVL C00054 +MOVJ EC00054
SMOVL C00055 +MOVJ EC00055
SMOVL C00056 +MOVJ EC00056
SMOVL C00057 +MOVJ EC00057
SMOVL C00058 +MOVJ EC00058
SMOVL C00059 +MOVJ EC00059
SMOVL C00060 +MOVJ EC00060
SMOVL C00061 +MOVJ EC00061
SMOVL C00062 +MOVJ EC00062
SMOVL C00063 +MOVJ EC00063
SMOVL C00064 +MOVJ EC00064
SMOVL C00065 +MOVJ EC00065
SMOVL C00066 +MOVJ EC00066
SMOVL C00067 +MOVJ EC00067
SMOVL C00068 +MOVJ EC00068
SMOVL C00069 +MOVJ EC00069
SMOVL C00070 +MOVJ EC00070
SMOVL C00071 +MOVJ EC00071
SMOVL C00072 +MOVJ EC00072
SMOVL C00073 +MOVJ EC00073
SMOVL C00074 +MOVJ EC00074
SMOVL C00075 +MOVJ EC00075
SMOVL C00076 +MOVJ EC00076
SMOVL C00077 +MOVJ EC00077
SMOVL C00078 +MOVJ EC00078
SMOVL C00079 +MOVJ EC00079
SMOVL C00080 +MOVJ EC00080
SMOVL C00081 +MOVJ EC00081
SMOVL C00082 +MOVJ EC00082
SMOVL C00083 +MOVJ EC00083
SMOVL C00084 +MOVJ EC00084
SMOVL C00085 +MOVJ EC00085
SMOVL C00086 +MOVJ EC00086
SMOVL C00087 +MOVJ EC00087
SMOVL C00088 +MOVJ EC00088
SMOVL C00089 +MOVJ EC00089
SMOVL C00090 +MOVJ EC00090
SMOVL C00091 +MOVJ EC00091
SMOVL C00092 +MOVJ EC00092
SMOVL C00093 +MOVJ EC00093
SMOVL C00094 +MOVJ EC00094
SMOVL C00095 +MOVJ EC00095
SMOVL C00096 +MOVJ EC00096
SMOVL C00097 +MOVJ EC00097
SMOVL C00098 +MOVJ EC00098
SMOVL C00099 +MOVJ EC00099
SMOVL C00100 +MOVJ EC00100
SMOVL C00101 +MOVJ EC00101
SMOVL C00102 +MOVJ EC00102
SMOVL C00103 +MOVJ EC00103
SMOVL C00104 +MOVJ EC00104
SMOVL C00105 +MOVJ EC00105
SMOVL C00106 +MOVJ EC00106
SMOVL C00107 +MOVJ EC00107
SMOVL C00108 +MOVJ EC00108
SMOVL C00109 +MOVJ EC00109
SMOVL C00110 +MOVJ EC00110
SMOVL C00111 +MOVJ EC00111
SMOVL C00112 +MOVJ EC00112
SMOVL C00113 +MOVJ EC00113
SMOVL C00114 +MOVJ EC00114
SMOVL C00115 +MOVJ EC00115
SMOVL C00116 +MOVJ EC00116
SMOVL C00117 +MOVJ EC00117
SMOVL C00118 +MOVJ EC00118
SMOVL C00119 +MOVJ EC00119
SMOVL C00120 +MOVJ EC00120
SMOVL C00121 +MOVJ EC00121
SMOVL C00122 +MOVJ EC00122
SMOVL C00123 +MOVJ EC00123
SMOVL C00124 +MOVJ EC00124
SMOVL C00125 +MOVJ EC00125
SMOVL C00126 +MOVJ EC00126
SMOVL C00127 +MOVJ EC00127
SMOVL C00128 +MOVJ EC00128
SMOVL C00129 +MOVJ EC00129
SMOVL C00130 +MOVJ EC00130
SMOVL C00131 +MOVJ EC00131
SMOVL C00132 +MOVJ EC00132
SMOVL C00133 +MOVJ EC00133
SMOVL C00134 +MOVJ EC00134
SMOVL C00135 +MOVJ EC00135
SMOVL C00136 +MOVJ EC00136
SMOVL C00137 +MOVJ EC00137
SMOVL C00138 +MOVJ EC00138
SMOVL C00139 +MOVJ EC00139
SMOVL C00140 +MOVJ EC00140
SMOVL C00141 +MOVJ EC00141
SMOVL C00142 +MOVJ EC00142
SMOVL C00143 +MOVJ EC00143
SMOVL C00144 +MOVJ EC00144
SMOVL C00145 +MOVJ EC00145
SMOVL C00146 +MOVJ EC00146
SMOVL C00147 +MOVJ EC00147
SMOVL C00148 +MOVJ EC00148
SMOVL C00149 +MOVJ EC00149
SMOVL C00150 +MOVJ EC00150
SMOVL C00151 +MOVJ EC00151
SMOVL C00152 +MOVJ EC00152
SMOVL C00153 +MOVJ EC00153
SMOVL C00154 +MOVJ EC00154
SMOVL C00155 +MOVJ EC00155
SMOVL C00156 +MOVJ EC00156
SMOVL C00157 +MOVJ EC00157
SMOVL C00158 +MOVJ EC00158
SMOVL C00159 +MOVJ EC00159
SMOVL C00160 +MOVJ EC00160
SMOVL C00161 +MOVJ EC00161
SMOVL C00162 +MOVJ EC00162
SMOVL C00163 +MOVJ EC00163
SMOVL C00164 +MOVJ EC00164
SMOVL C00165 +MOVJ EC00165
SMOVL C00166 +MOVJ EC00166
SMOVL C00167 +MOVJ EC00167
SMOVL C00168 +MOVJ EC00168
SMOVL C00169 +MOVJ EC00169
SMOVL C00170 +MOVJ EC00170
SMOVL C00171 +MOVJ EC00171
SMOVL C00172 +MOVJ EC00172
SMOVL C00173 +MOVJ EC00173
SMOVL C00174 +MOVJ EC00174
SMOVL C00175 +MOVJ EC00175
SMOVL C00176 +MOVJ EC00176
SMOVL C00177 +MOVJ EC00177
SMOVL C00178 +MOVJ EC00178
SMOVL C00179 +MOVJ EC00179
SMOVL C00180 +MOVJ EC00180
SMOVL C00181 +MOVJ EC00181
SMOVL C00182 +MOVJ EC00182
SMOVL C00183 +MOVJ EC00183
SMOVL C00184 +MOVJ EC00184
SMOVL C00185 +MOVJ EC00185
SMOVL C00186 +MOVJ EC00186
SMOVL C00187 +MOVJ EC00187
SMOVL C00188 +MOVJ EC00188
SMOVL C00189 +MOVJ EC00189
SMOVL C00190 +MOVJ EC00190
SMOVL C00191 +MOVJ EC00191
SMOVL C00192 +MOVJ EC00192
SMOVL C00193 +MOVJ EC00193
SMOVL C00194 +MOVJ EC00194
SMOVL C00195 +MOVJ EC00195
SMOVL C00196 +MOVJ EC00196
SMOVL C00197 +MOVJ EC00197
SMOVL C00198 +MOVJ EC00198
SMOVL C00199 +MOVJ EC00199
SMOVL C00200 +MOVJ EC00200
SMOVL C00201 +MOVJ EC00201
SMOVL C00202 +MOVJ EC00202
SMOVL C00203 +MOVJ EC00203
SMOVL C00204 +MOVJ EC00204
SMOVL C00205 +MOVJ EC00205
SMOVL C00206 +MOVJ EC00206
SMOVL C00207 +MOVJ EC00207
SMOVL C00208 +MOVJ EC00208
SMOVL C00209 +MOVJ EC00209
SMOVL C00210 +MOVJ EC00210
SMOVL C00211 +MOVJ EC00211
SMOVL C00212 +MOVJ EC00212
SMOVL C00213 +MOVJ EC00213
SMOVL C00214 +MOVJ EC00214
SMOVL C00215 +MOVJ EC00215
SMOVL C00216 +MOVJ EC00216
SMOVL C00217 +MOVJ EC00217
SMOVL C00218 +MOVJ EC00218
SMOVL C00219 +MOVJ EC00219
SMOVL C00220 +MOVJ EC00220
SMOVL C00221 +MOVJ EC00221
SMOVL C00222 +MOVJ EC00222
SMOVL C00223 +MOVJ EC00223
SMOVL C00224 +MOVJ EC00224
SMOVL C00225 +MOVJ EC00225
SMOVL C00226 +MOVJ EC00226
SMOVL C00227 +MOVJ EC00227
SMOVL C00228 +MOVJ EC00228
SMOVL C00229 +MOVJ EC00229
SMOVL C00230 +MOVJ EC00230
SMOVL C00231 +MOVJ EC00231
SMOVL C00232 +MOVJ EC00232
SMOVL C00233 +MOVJ EC00233
SMOVL C00234 +MOVJ EC00234
SMOVL C00235 +MOVJ EC00235
SMOVL C00236 +MOVJ EC00236
SMOVL C00237 +MOVJ EC00237
SMOVL C00238 +MOVJ EC00238
SMOVL C00239 +MOVJ EC00239
SMOVL C00240 +MOVJ EC00240
SMOVL C00241 +MOVJ EC00241
SMOVL C00242 +MOVJ EC00242
SMOVL C00243 +MOVJ EC00243
SMOVL C00244 +MOVJ EC00244
SMOVL C00245 +MOVJ EC00245
SMOVL C00246 +MOVJ EC00246
SMOVL C00247 +MOVJ EC00247
SMOVL C00248 +MOVJ EC00248
SMOVL C00249 +MOVJ EC00249
SMOVL C00250 +MOVJ EC00250
SMOVL C00251 +MOVJ EC00251
SMOVL C00252 +MOVJ EC00252
SMOVL C00253 +MOVJ EC00253
SMOVL C00254 +MOVJ EC00254
SMOVL C00255 +MOVJ EC00255
SMOVL C00256 +MOVJ EC00256
SMOVL C00257 +MOVJ EC00257
SMOVL C00258 +MOVJ EC00258
SMOVL C00259 +MOVJ EC00259
SMOVL C00260 +MOVJ EC00260
SMOVL C00261 +MOVJ EC00261
SMOVL C00262 +MOVJ EC00262
SMOVL C00263 +MOVJ EC00263
SMOVL C00264 +MOVJ EC00264
SMOVL C00265 +MOVJ EC00265
SMOVL C00266 +MOVJ EC00266
SMOVL C00267 +MOVJ EC00267
SMOVL C00268 +MOVJ EC00268
SMOVL C00269 +MOVJ EC00269
SMOVL C00270 +MOVJ EC00270
SMOVL C00271 +MOVJ EC00271
SMOVL C00272 +MOVJ EC00272
SMOVL C00273 +MOVJ EC00273
SMOVL C00274 +MOVJ EC00274
SMOVL C00275 +MOVJ EC00275
SMOVL C00276 +MOVJ EC00276
SMOVL C00277 +MOVJ EC00277
SMOVL C00278 +MOVJ EC00278
SMOVL C00279 +MOVJ EC00279
SMOVL C00280 +MOVJ EC00280
SMOVL C00281 +MOVJ EC00281
SMOVL C00282 +MOVJ EC00282
SMOVL C00283 +MOVJ EC00283
SMOVL C00284 +MOVJ EC00284
SMOVL C00285 +MOVJ EC00285
SMOVL C00286 +MOVJ EC00286
SMOVL C00287 +MOVJ EC00287
SMOVL C00288 +MOVJ EC00288
SMOVL C00289 +MOVJ EC00289
SMOVL C00290 +MOVJ EC00290
SMOVL C00291 +MOVJ EC00291
SMOVL C00292 +MOVJ EC00292
SMOVL C00293 +MOVJ EC00293
SMOVL C00294 +MOVJ EC00294
SMOVL C00295 +MOVJ EC00295
SMOVL C00296 +MOVJ EC00296
SMOVL C00297 +MOVJ EC00297
SMOVL C00298 +MOVJ EC00298
SMOVL C00299 +MOVJ EC00299
SMOVL C00300 +MOVJ EC00300
SMOVL C00301 +MOVJ EC00301
SMOVL C00302 +MOVJ EC00302
SMOVL C00303 +MOVJ EC00303
SMOVL C00304 +MOVJ EC00304
SMOVL C00305 +MOVJ EC00305
SMOVL C00306 +MOVJ EC00306
SMOVL C00307 +MOVJ EC00307
SMOVL C00308 +MOVJ EC00308
SMOVL C00309 +MOVJ EC00309
SMOVL C00310 +MOVJ EC00310
SMOVL C00311 +MOVJ EC00311
SMOVL C00312 +MOVJ EC00312
SMOVL C00313 +MOVJ EC00313
SMOVL C00314 +MOVJ EC00314
SMOVL C00315 +MOVJ EC00315
SMOVL C00316 +MOVJ EC00316
SMOVL C00317 +MOVJ EC00317
SMOVL C00318 +MOVJ EC00318
SMOVL C00319 +MOVJ EC00319
SMOVL C00320 +MOVJ EC00320
SMOVL C00321 +MOVJ EC00321
SMOVL C00322 +MOVJ EC00322
SMOVL C00323 +MOVJ EC00323
SMOVL C00324 +MOVJ EC00324
SMOVL C00325 +MOVJ EC00325
SMOVL C00326 +MOVJ EC00326
SMOVL C00327 +MOVJ EC00327
SMOVL C00328 +MOVJ EC00328
SMOVL C00329 +MOVJ EC00329
SMOVL C00330 +MOVJ EC00330
SMOVL C00331 +MOVJ EC00331
SMOVL C00332 +MOVJ EC00332
SMOVL C00333 +MOVJ EC00333
SMOVL C00334 +MOVJ EC00334
SMOVL C00335 +MOVJ EC00335
SMOVL C00336 +MOVJ EC00336
SMOVL C00337 +MOVJ EC00337
SMOVL C00338 +MOVJ EC00338
SMOVL C00339 +MOVJ EC00339
SMOVL C00340 +MOVJ EC00340
SMOVL C00341 +MOVJ EC00341
SMOVL C00342 +MOVJ EC00342
SMOVL C00343 +MOVJ EC00343
SMOVL C00344 +MOVJ EC00344
SMOVL C00345 +MOVJ EC00345
SMOVL C00346 +MOVJ EC00346
SMOVL C00347 +MOVJ EC00347
SMOVL C00348 +MOVJ EC00348
SMOVL C00349 +MOVJ EC00349
SMOVL C00350 +MOVJ EC00350
SMOVL C00351 +MOVJ EC00351
SMOVL C00352 +MOVJ EC00352
SMOVL C00353 +MOVJ EC00353
SMOVL C00354 +MOVJ EC00354
SMOVL C00355 +MOVJ EC00355
SMOVL C00356 +MOVJ EC00356
SMOVL C00357 +MOVJ EC00357
SMOVL C00358 +MOVJ EC00358
SMOVL C00359 +MOVJ EC00359
SMOVL C00360 +MOVJ EC00360
SMOVL C00361 +MOVJ EC00361
SMOVL C00362 +MOVJ EC00362
SMOVL C00363 +MOVJ EC00363
SMOVL C00364 +MOVJ EC00364
SMOVL C00365 +MOVJ EC00365
SMOVL C00366 +MOVJ EC00366
SMOVL C00367 +MOVJ EC00367
SMOVL C00368 +MOVJ EC00368
SMOVL C00369 +MOVJ EC00369
SMOVL C00370 +MOVJ EC00370
SMOVL C00371 +MOVJ EC00371
SMOVL C00372 +MOVJ EC00372
SMOVL C00373 +MOVJ EC00373
SMOVL C00374 +MOVJ EC00374
SMOVL C00375 +MOVJ EC00375
SMOVL C00376 +MOVJ EC00376
SMOVL C00377 +MOVJ EC00377
SMOVL C00378 +MOVJ EC00378
SMOVL C00379 +MOVJ EC00379
SMOVL C00380 +MOVJ EC00380
SMOVL C00381 +MOVJ EC00381
SMOVL C00382 +MOVJ EC00382
SMOVL C00383 +MOVJ EC00383
SMOVL C00384 +MOVJ EC00384
SMOVL C00385 +MOVJ EC00385
SMOVL C00386 +MOVJ EC00386
SMOVL C00387 +MOVJ EC00387
SMOVL C00388 +MOVJ EC00388
SMOVL C00389 +MOVJ EC00389
SMOVL C00390 +MOVJ EC00390
SMOVL C00391 +MOVJ EC00391
SMOVL C00392 +MOVJ EC00392
SMOVL C00393 +MOVJ EC00393
SMOVL C00394 +MOVJ EC00394
SMOVL C00395 +MOVJ EC00395
SMOVL C00396 +MOVJ EC00396
SMOVL C00397 +MOVJ EC00397
SMOVL C00398 +MOVJ EC00398
SMOVL C00399 +MOVJ EC00399
SMOVL C00400 +MOVJ EC00400
SMOVL C00401 +MOVJ EC00401
SMOVL C00402 +MOVJ EC00402
SMOVL C00403 +MOVJ EC00403
SMOVL C00404 +MOVJ EC00404
SMOVL C00405 +MOVJ EC00405
SMOVL C00406 +MOVJ EC00406
SMOVL C00407 +MOVJ EC00407
SMOVL C00408 +MOVJ EC00408
SMOVL C00409 +MOVJ EC00409
SMOVL C00410 +MOVJ EC00410
SMOVL C00411 +MOVJ EC00411
SMOVL C00412 +MOVJ EC00412
SMOVL C00413 +MOVJ EC00413
SMOVL C00414 +MOVJ EC00414
SMOVL C00415 +MOVJ EC00415
SMOVL C00416 +MOVJ EC00416
SMOVL C00417 +MOVJ EC00417
SMOVL C00418 +MOVJ EC00418
SMOVL C00419 +MOVJ EC00419
SMOVL C00420 +MOVJ EC00420
SMOVL C00421 +MOVJ EC00421
SMOVL C00422 +MOVJ EC00422
SMOVL C00423 +MOVJ EC00423
SMOVL C00424 +MOVJ EC00424
SMOVL C00425 +MOVJ EC00425
SMOVL C00426 +MOVJ EC00426
SMOVL C00427 +MOVJ EC00427
SMOVL C00428 +MOVJ EC00428
SMOVL C00429 +MOVJ EC00429
SMOVL C00430 +MOVJ EC00430
SMOVL C00431 +MOVJ EC00431
SMOVL C00432 +MOVJ EC00432
SMOVL C00433 +MOVJ EC00433
SMOVL C00434 +MOVJ EC00434
SMOVL C00435 +MOVJ EC00435
SMOVL C00436 +MOVJ EC00436
SMOVL C00437 +MOVJ EC00437
SMOVL C00438 +MOVJ EC00438
SMOVL C00439 +MOVJ EC00439
SMOVL C00440 +MOVJ EC00440
SMOVL C00441 +MOVJ EC00441
SMOVL C00442 +MOVJ EC00442
SMOVL C00443 +MOVJ EC00443
SMOVL C00444 +MOVJ EC00444
SMOVL C00445 +MOVJ EC00445
SMOVL C00446 +MOVJ EC00446
SMOVL C00447 +MOVJ EC00447
SMOVL C00448 +MOVJ EC00448
SMOVL C00449 +MOVJ EC00449
SMOVL C00450 +MOVJ EC00450
SMOVL C00451 +MOVJ EC00451
SMOVL C00452 +MOVJ EC00452
SMOVL C00453 +MOVJ EC00453
SMOVL C00454 +MOVJ EC00454
SMOVL C00455 +MOVJ EC00455
SMOVL C00456 +MOVJ EC00456
SMOVL C00457 +MOVJ EC00457
SMOVL C00458 +MOVJ EC00458
SMOVL C00459 +MOVJ EC00459
SMOVL C00460 +MOVJ EC00460
SMOVL C00461 +MOVJ EC00461
SMOVL C00462 +MOVJ EC00462
SMOVL C00463 +MOVJ EC00463
SMOVL C00464 +MOVJ EC00464
SMOVL C00465 +MOVJ EC00465
SMOVL C00466 +MOVJ EC00466
SMOVL C00467 +MOVJ EC00467
SMOVL C00468 +MOVJ EC00468
SMOVL C00469 +MOVJ EC00469
SMOVL C00470 +MOVJ EC00470
SMOVL C00471 +MOVJ EC00471
SMOVL C00472 +MOVJ EC00472
SMOVL C00473 +MOVJ EC00473
SMOVL C00474 +MOVJ EC00474
SMOVL C00475 +MOVJ EC00475
SMOVL C00476 +MOVJ EC00476
SMOVL C00477 +MOVJ EC00477
SMOVL C00478 +MOVJ EC00478
SMOVL C00479 +MOVJ EC00479
SMOVL C00480 +MOVJ EC00480
SMOVL C00481 +MOVJ EC00481
SMOVL C00482 +MOVJ EC00482
SMOVL C00483 +MOVJ EC00483
SMOVL C00484 +MOVJ EC00484
SMOVL C00485 +MOVJ EC00485
SMOVL C00486 +MOVJ EC00486
SMOVL C00487 +MOVJ EC00487
SMOVL C00488 +MOVJ EC00488
SMOVL C00489 +MOVJ EC00489
SMOVL C00490 +MOVJ EC00490
SMOVL C00491 +MOVJ EC00491
SMOVL C00492 +MOVJ EC00492
SMOVL C00493 +MOVJ EC00493
SMOVL C00494 +MOVJ EC00494
SMOVL C00495 +MOVJ EC00495
SMOVL C00496 +MOVJ EC00496
SMOVL C00497 +MOVJ EC00497
SMOVL C00498 +MOVJ EC00498
SMOVL C00499 +MOVJ EC00499
SMOVL C00500 +MOVJ EC00500
SMOVL C00501 +MOVJ EC00501
SMOVL C00502 +MOVJ EC00502
SMOVL C00503 +MOVJ EC00503
SMOVL C00504 +MOVJ EC00504
SMOVL C00505 +MOVJ EC00505
SMOVL C00506 +MOVJ EC00506
SMOVL C00507 +MOVJ EC00507
SMOVL C00508 +MOVJ EC00508
SMOVL C00509 +MOVJ EC00509
SMOVL C00510 +MOVJ EC00510
SMOVL C00511 +MOVJ EC00511
SMOVL C00512 +MOVJ EC00512
SMOVL C00513 +MOVJ EC00513
SMOVL C00514 +MOVJ EC00514
SMOVL C00515 +MOVJ EC00515
SMOVL C00516 +MOVJ EC00516
SMOVL C00517 +MOVJ EC00517
SMOVL C00518 +MOVJ EC00518
SMOVL C00519 +MOVJ EC00519
SMOVL C00520 +MOVJ EC00520
SMOVL C00521 +MOVJ EC00521
SMOVL C00522 +MOVJ EC00522
SMOVL C00523 +MOVJ EC00523
SMOVL C00524 +MOVJ EC00524
SMOVL C00525 +MOVJ EC00525
SMOVL C00526 +MOVJ EC00526
SMOVL C00527 +MOVJ EC00527
SMOVL C00528 +MOVJ EC00528
SMOVL C00529 +MOVJ EC00529
SMOVL C00530 +MOVJ EC00530
SMOVL C00531 +MOVJ EC00531
SMOVL C00532 +MOVJ EC00532
SMOVL C00533 +MOVJ EC00533
SMOVL C00534 +MOVJ EC00534
SMOVL C00535 +MOVJ EC00535
SMOVL C00536 +MOVJ EC00536
SMOVL C00537 +MOVJ EC00537
SMOVL C00538 +MOVJ EC00538
SMOVL C00539 +MOVJ EC00539
SMOVL C00540 +MOVJ EC00540
SMOVL C00541 +MOVJ EC00541
SMOVL C00542 +MOVJ EC00542
SMOVL C00543 +MOVJ EC00543
SMOVL C00544 +MOVJ EC00544
SMOVL C00545 +MOVJ EC00545
SMOVL C00546 +MOVJ EC00546
SMOVL C00547 +MOVJ EC00547
SMOVL C00548 +MOVJ EC00548
SMOVL C00549 +MOVJ EC00549
SMOVL C00550 +MOVJ EC00550
SMOVL C00551 +MOVJ EC00551
SMOVL C00552 +MOVJ EC00552
SMOVL C00553 +MOVJ EC00553
SMOVL C00554 +MOVJ EC00554
SMOVL C00555 +MOVJ EC00555
SMOVL C00556 +MOVJ EC00556
SMOVL C00557 +MOVJ EC00557
SMOVL C00558 +MOVJ EC00558
SMOVL C00559 +MOVJ EC00559
SMOVL C00560 +MOVJ EC00560
SMOVL C00561 +MOVJ EC00561
SMOVL C00562 +MOVJ EC00562
SMOVL C00563 +MOVJ EC00563
SMOVL C00564 +MOVJ EC00564
SMOVL C00565 +MOVJ EC00565
SMOVL C00566 +MOVJ EC00566
SMOVL C00567 +MOVJ EC00567
SMOVL C00568 +MOVJ EC00568
SMOVL C00569 +MOVJ EC00569
SMOVL C00570 +MOVJ EC00570
SMOVL C00571 +MOVJ EC00571
SMOVL C00572 +MOVJ EC00572
SMOVL C00573 +MOVJ EC00573
SMOVL C00574 +MOVJ EC00574
SMOVL C00575 +MOVJ EC00575
SMOVL C00576 +MOVJ EC00576
SMOVL C00577 +MOVJ EC00577
SMOVL C00578 +MOVJ EC00578
SMOVL C00579 +MOVJ EC00579
SMOVL C00580 +MOVJ EC00580
SMOVL C00581 +MOVJ EC00581
SMOVL C00582 +MOVJ EC00582
SMOVL C00583 +MOVJ EC00583
SMOVL C00584 +MOVJ EC00584
SMOVL C00585 +MOVJ EC00585
SMOVL C00586 +MOVJ EC00586
SMOVL C00587 +MOVJ EC00587
SMOVL C00588 +MOVJ EC00588
SMOVL C00589 +MOVJ EC00589
SMOVL C00590 +MOVJ EC00590
SMOVL C00591 +MOVJ EC00591
SMOVL C00592 +MOVJ EC00592
SMOVL C00593 +MOVJ EC00593
SMOVL C00594 +MOVJ EC00594
SMOVL C00595 +MOVJ EC00595
SMOVL C00596 +MOVJ EC00596
SMOVL C00597 +MOVJ EC00597
SMOVL C00598 +MOVJ EC00598
SMOVL C00599 +MOVJ EC00599
SMOVL C00600 +MOVJ EC00600
SMOVL C00601 +MOVJ EC00601
SMOVL C00602 +MOVJ EC00602
SMOVL C00603 +MOVJ EC00603
SMOVL C00604 +MOVJ EC00604
SMOVL C00605 +MOVJ EC00605
SMOVL C00606 +MOVJ EC00606
SMOVL C00607 +MOVJ EC00607
SMOVL C00608 +MOVJ EC00608
SMOVL C00609 +MOVJ EC00609
SMOVL C00610 +MOVJ EC00610
SMOVL C00611 +MOVJ EC00611
SMOVL C00612 +MOVJ EC00612
SMOVL C00613 +MOVJ EC00613
SMOVL C00614 +MOVJ EC00614
SMOVL C00615 +MOVJ EC00615
SMOVL C00616 +MOVJ EC00616
SMOVL C00617 +MOVJ EC00617
SMOVL C00618 +MOVJ EC00618
SMOVL C00619 +MOVJ EC00619
SMOVL C00620 +MOVJ EC00620
SMOVL C00621 +MOVJ EC00621
SMOVL C00622 +MOVJ EC00622
SMOVL C00623 +MOVJ EC00623
SMOVL C00624 +MOVJ EC00624
SMOVL C00625 +MOVJ EC00625
SMOVL C00626 +MOVJ EC00626
SMOVL C00627 +MOVJ EC00627
SMOVL C00628 +MOVJ EC00628
SMOVL C00629 +MOVJ EC00629
SMOVL C00630 +MOVJ EC00630
SMOVL C00631 +MOVJ EC00631
SMOVL C00632 +MOVJ EC00632
SMOVL C00633 +MOVJ EC00633
SMOVL C00634 +MOVJ EC00634
SMOVL C00635 +MOVJ EC00635
SMOVL C00636 +MOVJ EC00636
SMOVL C00637 +MOVJ EC00637
SMOVL C00638 +MOVJ EC00638
SMOVL C00639 +MOVJ EC00639
SMOVL C00640 +MOVJ EC00640
SMOVL C00641 +MOVJ EC00641
SMOVL C00642 +MOVJ EC00642
SMOVL C00643 +MOVJ EC00643
SMOVL C00644 +MOVJ EC00644
SMOVL C00645 +MOVJ EC00645
SMOVL C00646 +MOVJ EC00646
SMOVL C00647 +MOVJ EC00647
SMOVL C00648 +MOVJ EC00648
SMOVL C00649 +MOVJ EC00649
SMOVL C00650 +MOVJ EC00650
SMOVL C00651 +MOVJ EC00651
SMOVL C00652 +MOVJ EC00652
SMOVL C00653 +MOVJ EC00653
SMOVL C00654 +MOVJ EC00654
SMOVL C00655 +MOVJ EC00655
SMOVL C00656 +MOVJ EC00656
SMOVL C00657 +MOVJ EC00657
SMOVL C00658 +MOVJ EC00658
SMOVL C00659 +MOVJ EC00659
SMOVL C00660 +MOVJ EC00660
SMOVL C00661 +MOVJ EC00661
SMOVL C00662 +MOVJ EC00662
SMOVL C00663 +MOVJ EC00663
SMOVL C00664 +MOVJ EC00664
SMOVL C00665 +MOVJ EC00665
SMOVL C00666 +MOVJ EC00666
SMOVL C00667 +MOVJ EC00667
SMOVL C00668 +MOVJ EC00668
SMOVL C00669 +MOVJ EC00669
SMOVL C00670 +MOVJ EC00670
SMOVL C00671 +MOVJ EC00671
SMOVL C00672 +MOVJ EC00672
SMOVL C00673 +MOVJ EC00673
SMOVL C00674 +MOVJ EC00674
SMOVL C00675 +MOVJ EC00675
SMOVL C00676 +MOVJ EC00676
SMOVL C00677 +MOVJ EC00677
SMOVL C00678 +MOVJ EC00678
SMOVL C00679 +MOVJ EC00679
SMOVL C00680 +MOVJ EC00680
SMOVL C00681 +MOVJ EC00681
SMOVL C00682 +MOVJ EC00682
SMOVL C00683 +MOVJ EC00683
SMOVL C00684 +MOVJ EC00684
SMOVL C00685 +MOVJ EC00685
SMOVL C00686 +MOVJ EC00686
SMOVL C00687 +MOVJ EC00687
SMOVL C00688 +MOVJ EC00688
SMOVL C00689 +MOVJ EC00689
SMOVL C00690 +MOVJ EC00690
SMOVL C00691 +MOVJ EC00691
SMOVL C00692 +MOVJ EC00692
SMOVL C00693 +MOVJ EC00693
SMOVL C00694 +MOVJ EC00694
SMOVL C00695 +MOVJ EC00695
SMOVL C00696 +MOVJ EC00696
SMOVL C00697 +MOVJ EC00697
SMOVL C00698 +MOVJ EC00698
SMOVL C00699 +MOVJ EC00699
SMOVL C00700 +MOVJ EC00700
SMOVL C00701 +MOVJ EC00701
SMOVL C00702 +MOVJ EC00702
SMOVL C00703 +MOVJ EC00703
SMOVL C00704 +MOVJ EC00704
SMOVL C00705 +MOVJ EC00705
SMOVL C00706 +MOVJ EC00706
SMOVL C00707 +MOVJ EC00707
SMOVL C00708 +MOVJ EC00708
SMOVL C00709 +MOVJ EC00709
SMOVL C00710 +MOVJ EC00710
SMOVL C00711 +MOVJ EC00711
SMOVL C00712 +MOVJ EC00712
SMOVL C00713 +MOVJ EC00713
SMOVL C00714 +MOVJ EC00714
SMOVL C00715 +MOVJ EC00715
SMOVL C00716 +MOVJ EC00716
SMOVL C00717 +MOVJ EC00717
SMOVL C00718 +MOVJ EC00718
SMOVL C00719 +MOVJ EC00719
SMOVL C00720 +MOVJ EC00720
SMOVL C00721 +MOVJ EC00721
SMOVL C00722 +MOVJ EC00722
SMOVL C00723 +MOVJ EC00723
SMOVL C00724 +MOVJ EC00724
SMOVL C00725 +MOVJ EC00725
SMOVL C00726 +MOVJ EC00726
SMOVL C00727 +MOVJ EC00727
SMOVL C00728 +MOVJ EC00728
SMOVL C00729 +MOVJ EC00729
SMOVL C00730 +MOVJ EC00730
SMOVL C00731 +MOVJ EC00731
SMOVL C00732 +MOVJ EC00732
SMOVL C00733 +MOVJ EC00733
SMOVL C00734 +MOVJ EC00734
SMOVL C00735 +MOVJ EC00735
SMOVL C00736 +MOVJ EC00736
SMOVL C00737 +MOVJ EC00737
SMOVL C00738 +MOVJ EC00738
SMOVL C00739 +MOVJ EC00739
SMOVL C00740 +MOVJ EC00740
SMOVL C00741 +MOVJ EC00741
SMOVL C00742 +MOVJ EC00742
SMOVL C00743 +MOVJ EC00743
SMOVL C00744 +MOVJ EC00744
SMOVL C00745 +MOVJ EC00745
SMOVL C00746 +MOVJ EC00746
SMOVL C00747 +MOVJ EC00747
SMOVL C00748 +MOVJ EC00748
SMOVL C00749 +MOVJ EC00749
SMOVL C00750 +MOVJ EC00750
SMOVL C00751 +MOVJ EC00751
SMOVL C00752 +MOVJ EC00752
SMOVL C00753 +MOVJ EC00753
SMOVL C00754 +MOVJ EC00754
SMOVL C00755 +MOVJ EC00755
SMOVL C00756 +MOVJ EC00756
SMOVL C00757 +MOVJ EC00757
SMOVL C00758 +MOVJ EC00758
SMOVL C00759 +MOVJ EC00759
SMOVL C00760 +MOVJ EC00760
SMOVL C00761 +MOVJ EC00761
SMOVL C00762 +MOVJ EC00762
SMOVL C00763 +MOVJ EC00763
SMOVL C00764 +MOVJ EC00764
SMOVL C00765 +MOVJ EC00765
SMOVL C00766 +MOVJ EC00766
SMOVL C00767 +MOVJ EC00767
SMOVL C00768 +MOVJ EC00768
SMOVL C00769 +MOVJ EC00769
SMOVL C00770 +MOVJ EC00770
SMOVL C00771 +MOVJ EC00771
SMOVL C00772 +MOVJ EC00772
SMOVL C00773 +MOVJ EC00773
SMOVL C00774 +MOVJ EC00774
SMOVL C00775 +MOVJ EC00775
SMOVL C00776 +MOVJ EC00776
SMOVL C00777 +MOVJ EC00777
SMOVL C00778 +MOVJ EC00778
SMOVL C00779 +MOVJ EC00779
SMOVL C00780 +MOVJ EC00780
SMOVL C00781 +MOVJ EC00781
SMOVL C00782 +MOVJ EC00782
SMOVL C00783 +MOVJ EC00783
SMOVL C00784 +MOVJ EC00784
SMOVL C00785 +MOVJ EC00785
SMOVL C00786 +MOVJ EC00786
SMOVL C00787 +MOVJ EC00787
SMOVL C00788 +MOVJ EC00788
SMOVL C00789 +MOVJ EC00789
SMOVL C00790 +MOVJ EC00790
SMOVL C00791 +MOVJ EC00791
SMOVL C00792 +MOVJ EC00792
SMOVL C00793 +MOVJ EC00793
SMOVL C00794 +MOVJ EC00794
SMOVL C00795 +MOVJ EC00795
SMOVL C00796 +MOVJ EC00796
SMOVL C00797 +MOVJ EC00797
SMOVL C00798 +MOVJ EC00798
SMOVL C00799 +MOVJ EC00799
SMOVL C00800 +MOVJ EC00800
SMOVL C00801 +MOVJ EC00801
SMOVL C00802 +MOVJ EC00802
SMOVL C00803 +MOVJ EC00803
SMOVL C00804 +MOVJ EC00804
SMOVL C00805 +MOVJ EC00805
SMOVL C00806 +MOVJ EC00806
SMOVL C00807 +MOVJ EC00807
SMOVL C00808 +MOVJ EC00808
SMOVL C00809 +MOVJ EC00809
SMOVL C00810 +MOVJ EC00810
SMOVL C00811 +MOVJ EC00811
SMOVL C00812 +MOVJ EC00812
SMOVL C00813 +MOVJ EC00813
SMOVL C00814 +MOVJ EC00814
SMOVL C00815 +MOVJ EC00815
SMOVL C00816 +MOVJ EC00816
SMOVL C00817 +MOVJ EC00817
SMOVL C00818 +MOVJ EC00818
SMOVL C00819 +MOVJ EC00819
SMOVL C00820 +MOVJ EC00820
SMOVL C00821 +MOVJ EC00821
SMOVL C00822 +MOVJ EC00822
SMOVL C00823 +MOVJ EC00823
SMOVL C00824 +MOVJ EC00824
SMOVL C00825 +MOVJ EC00825
SMOVL C00826 +MOVJ EC00826
SMOVL C00827 +MOVJ EC00827
SMOVL C00828 +MOVJ EC00828
SMOVL C00829 +MOVJ EC00829
SMOVL C00830 +MOVJ EC00830
SMOVL C00831 +MOVJ EC00831
SMOVL C00832 +MOVJ EC00832
SMOVL C00833 +MOVJ EC00833
SMOVL C00834 +MOVJ EC00834
SMOVL C00835 +MOVJ EC00835
SMOVL C00836 +MOVJ EC00836
SMOVL C00837 +MOVJ EC00837
SMOVL C00838 +MOVJ EC00838
SMOVL C00839 +MOVJ EC00839
SMOVL C00840 +MOVJ EC00840
SMOVL C00841 +MOVJ EC00841
SMOVL C00842 +MOVJ EC00842
SMOVL C00843 +MOVJ EC00843
SMOVL C00844 +MOVJ EC00844
SMOVL C00845 +MOVJ EC00845
SMOVL C00846 +MOVJ EC00846
SMOVL C00847 +MOVJ EC00847
SMOVL C00848 +MOVJ EC00848
SMOVL C00849 +MOVJ EC00849
SMOVL C00850 +MOVJ EC00850
SMOVL C00851 +MOVJ EC00851
SMOVL C00852 +MOVJ EC00852
SMOVL C00853 +MOVJ EC00853
SMOVL C00854 +MOVJ EC00854
SMOVL C00855 +MOVJ EC00855
SMOVL C00856 +MOVJ EC00856
SMOVL C00857 +MOVJ EC00857
SMOVL C00858 +MOVJ EC00858
SMOVL C00859 +MOVJ EC00859
SMOVL C00860 +MOVJ EC00860
SMOVL C00861 +MOVJ EC00861
SMOVL C00862 +MOVJ EC00862
SMOVL C00863 +MOVJ EC00863
SMOVL C00864 +MOVJ EC00864
SMOVL C00865 +MOVJ EC00865
SMOVL C00866 +MOVJ EC00866
SMOVL C00867 +MOVJ EC00867
SMOVL C00868 +MOVJ EC00868
SMOVL C00869 +MOVJ EC00869
SMOVL C00870 +MOVJ EC00870
SMOVL C00871 +MOVJ EC00871
SMOVL C00872 +MOVJ EC00872
SMOVL C00873 +MOVJ EC00873
SMOVL C00874 +MOVJ EC00874
SMOVL C00875 +MOVJ EC00875
SMOVL C00876 +MOVJ EC00876
SMOVL C00877 +MOVJ EC00877
SMOVL C00878 +MOVJ EC00878
SMOVL C00879 +MOVJ EC00879
SMOVL C00880 +MOVJ EC00880
SMOVL C00881 +MOVJ EC00881
SMOVL C00882 +MOVJ EC00882
SMOVL C00883 +MOVJ EC00883
SMOVL C00884 +MOVJ EC00884
SMOVL C00885 +MOVJ EC00885
SMOVL C00886 +MOVJ EC00886
SMOVL C00887 +MOVJ EC00887
SMOVL C00888 +MOVJ EC00888
SMOVL C00889 +MOVJ EC00889
SMOVL C00890 +MOVJ EC00890
SMOVL C00891 +MOVJ EC00891
SMOVL C00892 +MOVJ EC00892
SMOVL C00893 +MOVJ EC00893
SMOVL C00894 +MOVJ EC00894
SMOVL C00895 +MOVJ EC00895
SMOVL C00896 +MOVJ EC00896
SMOVL C00897 +MOVJ EC00897
SMOVL C00898 +MOVJ EC00898
SMOVL C00899 +MOVJ EC00899
SMOVL C00900 +MOVJ EC00900
SMOVL C00901 +MOVJ EC00901
SMOVL C00902 +MOVJ EC00902
SMOVL C00903 +MOVJ EC00903
SMOVL C00904 +MOVJ EC00904
SMOVL C00905 +MOVJ EC00905
SMOVL C00906 +MOVJ EC00906
SMOVL C00907 +MOVJ EC00907
SMOVL C00908 +MOVJ EC00908
SMOVL C00909 +MOVJ EC00909
SMOVL C00910 +MOVJ EC00910
SMOVL C00911 +MOVJ EC00911
SMOVL C00912 +MOVJ EC00912
SMOVL C00913 +MOVJ EC00913
SMOVL C00914 +MOVJ EC00914
SMOVL C00915 +MOVJ EC00915
SMOVL C00916 +MOVJ EC00916
SMOVL C00917 +MOVJ EC00917
SMOVL C00918 +MOVJ EC00918
SMOVL C00919 +MOVJ EC00919
SMOVL C00920 +MOVJ EC00920
SMOVL C00921 +MOVJ EC00921
SMOVL C00922 +MOVJ EC00922
SMOVL C00923 +MOVJ EC00923
SMOVL C00924 +MOVJ EC00924
SMOVL C00925 +MOVJ EC00925
SMOVL C00926 +MOVJ EC00926
SMOVL C00927 +MOVJ EC00927
SMOVL C00928 +MOVJ EC00928
SMOVL C00929 +MOVJ EC00929
SMOVL C00930 +MOVJ EC00930
SMOVL C00931 +MOVJ EC00931
SMOVL C00932 +MOVJ EC00932
SMOVL C00933 +MOVJ EC00933
SMOVL C00934 +MOVJ EC00934
SMOVL C00935 +MOVJ EC00935
SMOVL C00936 +MOVJ EC00936
SMOVL C00937 +MOVJ EC00937
SMOVL C00938 +MOVJ EC00938
SMOVL C00939 +MOVJ EC00939
SMOVL C00940 +MOVJ EC00940
SMOVL C00941 +MOVJ EC00941
SMOVL C00942 +MOVJ EC00942
SMOVL C00943 +MOVJ EC00943
SMOVL C00944 +MOVJ EC00944
SMOVL C00945 +MOVJ EC00945
SMOVL C00946 +MOVJ EC00946
SMOVL C00947 +MOVJ EC00947
SMOVL C00948 +MOVJ EC00948
SMOVL C00949 +MOVJ EC00949
SMOVL C00950 +MOVJ EC00950
SMOVL C00951 +MOVJ EC00951
SMOVL C00952 +MOVJ EC00952
SMOVL C00953 +MOVJ EC00953
SMOVL C00954 +MOVJ EC00954
SMOVL C00955 +MOVJ EC00955
SMOVL C00956 +MOVJ EC00956
SMOVL C00957 +MOVJ EC00957
SMOVL C00958 +MOVJ EC00958
SMOVL C00959 +MOVJ EC00959
SMOVL C00960 +MOVJ EC00960
SMOVL C00961 +MOVJ EC00961
SMOVL C00962 +MOVJ EC00962
SMOVL C00963 +MOVJ EC00963
SMOVL C00964 +MOVJ EC00964
SMOVL C00965 +MOVJ EC00965
SMOVL C00966 +MOVJ EC00966
SMOVL C00967 +MOVJ EC00967
SMOVL C00968 +MOVJ EC00968
SMOVL C00969 +MOVJ EC00969
SMOVL C00970 +MOVJ EC00970
SMOVL C00971 +MOVJ EC00971
SMOVL C00972 +MOVJ EC00972
SMOVL C00973 +MOVJ EC00973
SMOVL C00974 +MOVJ EC00974
SMOVL C00975 +MOVJ EC00975
SMOVL C00976 +MOVJ EC00976
SMOVL C00977 +MOVJ EC00977
SMOVL C00978 +MOVJ EC00978
SMOVL C00979 +MOVJ EC00979
SMOVL C00980 +MOVJ EC00980
SMOVL C00981 +MOVJ EC00981
SMOVL C00982 +MOVJ EC00982
SMOVL C00983 +MOVJ EC00983
SMOVL C00984 +MOVJ EC00984
SMOVL C00985 +MOVJ EC00985
SMOVL C00986 +MOVJ EC00986
SMOVL C00987 +MOVJ EC00987
SMOVL C00988 +MOVJ EC00988
SMOVL C00989 +MOVJ EC00989
SMOVL C00990 +MOVJ EC00990
SMOVL C00991 +MOVJ EC00991
SMOVL C00992 +MOVJ EC00992
SMOVL C00993 +MOVJ EC00993
SMOVL C00994 +MOVJ EC00994
SMOVL C00995 +MOVJ EC00995
SMOVL C00996 +MOVJ EC00996
SMOVL C00997 +MOVJ EC00997
SMOVL C00998 +MOVJ EC00998
SMOVL C00999 +MOVJ EC00999
SMOVL C01000 +MOVJ EC01000
SMOVL C01001 +MOVJ EC01001
SMOVL C01002 +MOVJ EC01002
SMOVL C01003 +MOVJ EC01003
SMOVL C01004 +MOVJ EC01004
SMOVL C01005 +MOVJ EC01005
SMOVL C01006 +MOVJ EC01006
SMOVL C01007 +MOVJ EC01007
SMOVL C01008 +MOVJ EC01008
SMOVL C01009 +MOVJ EC01009
SMOVL C01010 +MOVJ EC01010
SMOVL C01011 +MOVJ EC01011
SMOVL C01012 +MOVJ EC01012
SMOVL C01013 +MOVJ EC01013
SMOVL C01014 +MOVJ EC01014
SMOVL C01015 +MOVJ EC01015
SMOVL C01016 +MOVJ EC01016
SMOVL C01017 +MOVJ EC01017
SMOVL C01018 +MOVJ EC01018
SMOVL C01019 +MOVJ EC01019
SMOVL C01020 +MOVJ EC01020
SMOVL C01021 +MOVJ EC01021
SMOVL C01022 +MOVJ EC01022
SMOVL C01023 +MOVJ EC01023
SMOVL C01024 +MOVJ EC01024
SMOVL C01025 +MOVJ EC01025
SMOVL C01026 +MOVJ EC01026
SMOVL C01027 +MOVJ EC01027
SMOVL C01028 +MOVJ EC01028
SMOVL C01029 +MOVJ EC01029
SMOVL C01030 +MOVJ EC01030
SMOVL C01031 +MOVJ EC01031
SMOVL C01032 +MOVJ EC01032
SMOVL C01033 +MOVJ EC01033
SMOVL C01034 +MOVJ EC01034
SMOVL C01035 +MOVJ EC01035
SMOVL C01036 +MOVJ EC01036
SMOVL C01037 +MOVJ EC01037
SMOVL C01038 +MOVJ EC01038
SMOVL C01039 +MOVJ EC01039
SMOVL C01040 +MOVJ EC01040
SMOVL C01041 +MOVJ EC01041
SMOVL C01042 +MOVJ EC01042
SMOVL C01043 +MOVJ EC01043
SMOVL C01044 +MOVJ EC01044
SMOVL C01045 +MOVJ EC01045
SMOVL C01046 +MOVJ EC01046
SMOVL C01047 +MOVJ EC01047
SMOVL C01048 +MOVJ EC01048
SMOVL C01049 +MOVJ EC01049
SMOVL C01050 +MOVJ EC01050
SMOVL C01051 +MOVJ EC01051
SMOVL C01052 +MOVJ EC01052
SMOVL C01053 +MOVJ EC01053
SMOVL C01054 +MOVJ EC01054
SMOVL C01055 +MOVJ EC01055
SMOVL C01056 +MOVJ EC01056
SMOVL C01057 +MOVJ EC01057
SMOVL C01058 +MOVJ EC01058
SMOVL C01059 +MOVJ EC01059
SMOVL C01060 +MOVJ EC01060
SMOVL C01061 +MOVJ EC01061
SMOVL C01062 +MOVJ EC01062
SMOVL C01063 +MOVJ EC01063
SMOVL C01064 +MOVJ EC01064
SMOVL C01065 +MOVJ EC01065
SMOVL C01066 +MOVJ EC01066
SMOVL C01067 +MOVJ EC01067
SMOVL C01068 +MOVJ EC01068
SMOVL C01069 +MOVJ EC01069
SMOVL C01070 +MOVJ EC01070
SMOVL C01071 +MOVJ EC01071
SMOVL C01072 +MOVJ EC01072
SMOVL C01073 +MOVJ EC01073
SMOVL C01074 +MOVJ EC01074
SMOVL C01075 +MOVJ EC01075
SMOVL C01076 +MOVJ EC01076
SMOVL C01077 +MOVJ EC01077
SMOVL C01078 +MOVJ EC01078
SMOVL C01079 +MOVJ EC01079
SMOVL C01080 +MOVJ EC01080
SMOVL C01081 +MOVJ EC01081
SMOVL C01082 +MOVJ EC01082
SMOVL C01083 +MOVJ EC01083
SMOVL C01084 +MOVJ EC01084
SMOVL C01085 +MOVJ EC01085
SMOVL C01086 +MOVJ EC01086
SMOVL C01087 +MOVJ EC01087
SMOVL C01088 +MOVJ EC01088
SMOVL C01089 +MOVJ EC01089
SMOVL C01090 +MOVJ EC01090
SMOVL C01091 +MOVJ EC01091
SMOVL C01092 +MOVJ EC01092
SMOVL C01093 +MOVJ EC01093
SMOVL C01094 +MOVJ EC01094
SMOVL C01095 +MOVJ EC01095
SMOVL C01096 +MOVJ EC01096
SMOVL C01097 +MOVJ EC01097
SMOVL C01098 +MOVJ EC01098
SMOVL C01099 +MOVJ EC01099
SMOVL C01100 +MOVJ EC01100
SMOVL C01101 +MOVJ EC01101
SMOVL C01102 +MOVJ EC01102
SMOVL C01103 +MOVJ EC01103
SMOVL C01104 +MOVJ EC01104
SMOVL C01105 +MOVJ EC01105
SMOVL C01106 +MOVJ EC01106
SMOVL C01107 +MOVJ EC01107
SMOVL C01108 +MOVJ EC01108
SMOVL C01109 +MOVJ EC01109
SMOVL C01110 +MOVJ EC01110
SMOVL C01111 +MOVJ EC01111
SMOVL C01112 +MOVJ EC01112
SMOVL C01113 +MOVJ EC01113
SMOVL C01114 +MOVJ EC01114
SMOVL C01115 +MOVJ EC01115
SMOVL C01116 +MOVJ EC01116
SMOVL C01117 +MOVJ EC01117
SMOVL C01118 +MOVJ EC01118
SMOVL C01119 +MOVJ EC01119
SMOVL C01120 +MOVJ EC01120
SMOVL C01121 +MOVJ EC01121
SMOVL C01122 +MOVJ EC01122
SMOVL C01123 +MOVJ EC01123
SMOVL C01124 +MOVJ EC01124
SMOVL C01125 +MOVJ EC01125
SMOVL C01126 +MOVJ EC01126
SMOVL C01127 +MOVJ EC01127
SMOVL C01128 +MOVJ EC01128
SMOVL C01129 +MOVJ EC01129
SMOVL C01130 +MOVJ EC01130
SMOVL C01131 +MOVJ EC01131
SMOVL C01132 +MOVJ EC01132
SMOVL C01133 +MOVJ EC01133
SMOVL C01134 +MOVJ EC01134
SMOVL C01135 +MOVJ EC01135
SMOVL C01136 +MOVJ EC01136
SMOVL C01137 +MOVJ EC01137
SMOVL C01138 +MOVJ EC01138
SMOVL C01139 +MOVJ EC01139
SMOVL C01140 +MOVJ EC01140
SMOVL C01141 +MOVJ EC01141
SMOVL C01142 +MOVJ EC01142
SMOVL C01143 +MOVJ EC01143
SMOVL C01144 +MOVJ EC01144
SMOVL C01145 +MOVJ EC01145
SMOVL C01146 +MOVJ EC01146
SMOVL C01147 +MOVJ EC01147
SMOVL C01148 +MOVJ EC01148
SMOVL C01149 +MOVJ EC01149
SMOVL C01150 +MOVJ EC01150
SMOVL C01151 +MOVJ EC01151
SMOVL C01152 +MOVJ EC01152
SMOVL C01153 +MOVJ EC01153
SMOVL C01154 +MOVJ EC01154
SMOVL C01155 +MOVJ EC01155
SMOVL C01156 +MOVJ EC01156
SMOVL C01157 +MOVJ EC01157
SMOVL C01158 +MOVJ EC01158
SMOVL C01159 +MOVJ EC01159
SMOVL C01160 +MOVJ EC01160
SMOVL C01161 +MOVJ EC01161
SMOVL C01162 +MOVJ EC01162
SMOVL C01163 +MOVJ EC01163
SMOVL C01164 +MOVJ EC01164
SMOVL C01165 +MOVJ EC01165
SMOVL C01166 +MOVJ EC01166
SMOVL C01167 +MOVJ EC01167
SMOVL C01168 +MOVJ EC01168
SMOVL C01169 +MOVJ EC01169
SMOVL C01170 +MOVJ EC01170
SMOVL C01171 +MOVJ EC01171
SMOVL C01172 +MOVJ EC01172
SMOVL C01173 +MOVJ EC01173
SMOVL C01174 +MOVJ EC01174
SMOVL C01175 +MOVJ EC01175
SMOVL C01176 +MOVJ EC01176
SMOVL C01177 +MOVJ EC01177
SMOVL C01178 +MOVJ EC01178
SMOVL C01179 +MOVJ EC01179
SMOVL C01180 +MOVJ EC01180
SMOVL C01181 +MOVJ EC01181
SMOVL C01182 +MOVJ EC01182
SMOVL C01183 +MOVJ EC01183
SMOVL C01184 +MOVJ EC01184
SMOVL C01185 +MOVJ EC01185
SMOVL C01186 +MOVJ EC01186
SMOVL C01187 +MOVJ EC01187
SMOVL C01188 +MOVJ EC01188
SMOVL C01189 +MOVJ EC01189
SMOVL C01190 +MOVJ EC01190
SMOVL C01191 +MOVJ EC01191
SMOVL C01192 +MOVJ EC01192
SMOVL C01193 +MOVJ EC01193
SMOVL C01194 +MOVJ EC01194
SMOVL C01195 +MOVJ EC01195
SMOVL C01196 +MOVJ EC01196
SMOVL C01197 +MOVJ EC01197
SMOVL C01198 +MOVJ EC01198
SMOVL C01199 +MOVJ EC01199
SMOVL C01200 +MOVJ EC01200
SMOVL C01201 +MOVJ EC01201
SMOVL C01202 +MOVJ EC01202
SMOVL C01203 +MOVJ EC01203
SMOVL C01204 +MOVJ EC01204
SMOVL C01205 +MOVJ EC01205
SMOVL C01206 +MOVJ EC01206
SMOVL C01207 +MOVJ EC01207
SMOVL C01208 +MOVJ EC01208
SMOVL C01209 +MOVJ EC01209
SMOVL C01210 +MOVJ EC01210
SMOVL C01211 +MOVJ EC01211
SMOVL C01212 +MOVJ EC01212
SMOVL C01213 +MOVJ EC01213
SMOVL C01214 +MOVJ EC01214
SMOVL C01215 +MOVJ EC01215
SMOVL C01216 +MOVJ EC01216
SMOVL C01217 +MOVJ EC01217
SMOVL C01218 +MOVJ EC01218
SMOVL C01219 +MOVJ EC01219
SMOVL C01220 +MOVJ EC01220
SMOVL C01221 +MOVJ EC01221
SMOVL C01222 +MOVJ EC01222
SMOVL C01223 +MOVJ EC01223
SMOVL C01224 +MOVJ EC01224
SMOVL C01225 +MOVJ EC01225
SMOVL C01226 +MOVJ EC01226
SMOVL C01227 +MOVJ EC01227
SMOVL C01228 +MOVJ EC01228
SMOVL C01229 +MOVJ EC01229
SMOVL C01230 +MOVJ EC01230
SMOVL C01231 +MOVJ EC01231
SMOVL C01232 +MOVJ EC01232
SMOVL C01233 +MOVJ EC01233
SMOVL C01234 +MOVJ EC01234
SMOVL C01235 +MOVJ EC01235
SMOVL C01236 +MOVJ EC01236
SMOVL C01237 +MOVJ EC01237
SMOVL C01238 +MOVJ EC01238
SMOVL C01239 +MOVJ EC01239
SMOVL C01240 +MOVJ EC01240
SMOVL C01241 +MOVJ EC01241
SMOVL C01242 +MOVJ EC01242
SMOVL C01243 +MOVJ EC01243
SMOVL C01244 +MOVJ EC01244
SMOVL C01245 +MOVJ EC01245
SMOVL C01246 +MOVJ EC01246
SMOVL C01247 +MOVJ EC01247
SMOVL C01248 +MOVJ EC01248
SMOVL C01249 +MOVJ EC01249
SMOVL C01250 +MOVJ EC01250
SMOVL C01251 +MOVJ EC01251
SMOVL C01252 +MOVJ EC01252
SMOVL C01253 +MOVJ EC01253
SMOVL C01254 +MOVJ EC01254
SMOVL C01255 +MOVJ EC01255
SMOVL C01256 +MOVJ EC01256
SMOVL C01257 +MOVJ EC01257
SMOVL C01258 +MOVJ EC01258
SMOVL C01259 +MOVJ EC01259
SMOVL C01260 +MOVJ EC01260
SMOVL C01261 +MOVJ EC01261
SMOVL C01262 +MOVJ EC01262
SMOVL C01263 +MOVJ EC01263
SMOVL C01264 +MOVJ EC01264
SMOVL C01265 +MOVJ EC01265
SMOVL C01266 +MOVJ EC01266
SMOVL C01267 +MOVJ EC01267
SMOVL C01268 +MOVJ EC01268
SMOVL C01269 +MOVJ EC01269
SMOVL C01270 +MOVJ EC01270
SMOVL C01271 +MOVJ EC01271
SMOVL C01272 +MOVJ EC01272
SMOVL C01273 +MOVJ EC01273
SMOVL C01274 +MOVJ EC01274
